// TIA Portal V16 export
// export: Created 2024-05-17T05:47:00.9022411Z, ExportSetting WithDefaults, DisplayName Totally Integrated Automation Portal, DisplayVersion V16, DisplayName TIA Portal Version Control Interface, DisplayVersion V16, DisplayName TIA Portal Openness, DisplayVersion V16, DisplayName STEP 7 Professional, DisplayVersion V16, DisplayName STEP 7 Safety, DisplayVersion V16, DisplayName WinCC Professional, DisplayVersion V16
FUNCTION_BLOCK "K03_状态"   // FB3, LAD
{ S7_Optimized_Access := 'TRUE' }
VERSION : 0.1
// stored: AutoNumber false, IsIECCheckEnabled false, IsRetainMemResEnabled false, MemoryReserve 100, SetENOAutomatically false, UDAEnableTagReadback false
   VAR
      放行延迟 : IEC_TIMER;
   END_VAR
   VAR_TEMP
      M_Pluse : Array[1..20] of Bool;
   END_VAR
   VAR_TEMP   // added for the SCL form of the ladder/FBD networks
      _w1 : Bool;
      _w2 : Bool;
      _w3 : Bool;
      _w4 : Bool;
      _w5 : Bool;
      _w6 : Bool;
      _w7 : Bool;
      _w8 : Bool;
      _w9 : Bool;
      _w10 : Bool;
      _w11 : Bool;
      _w12 : Bool;
      _w13 : Bool;
      _w14 : Bool;
      _w15 : Bool;
   END_VAR
BEGIN

REGION Network 1: 初始2s
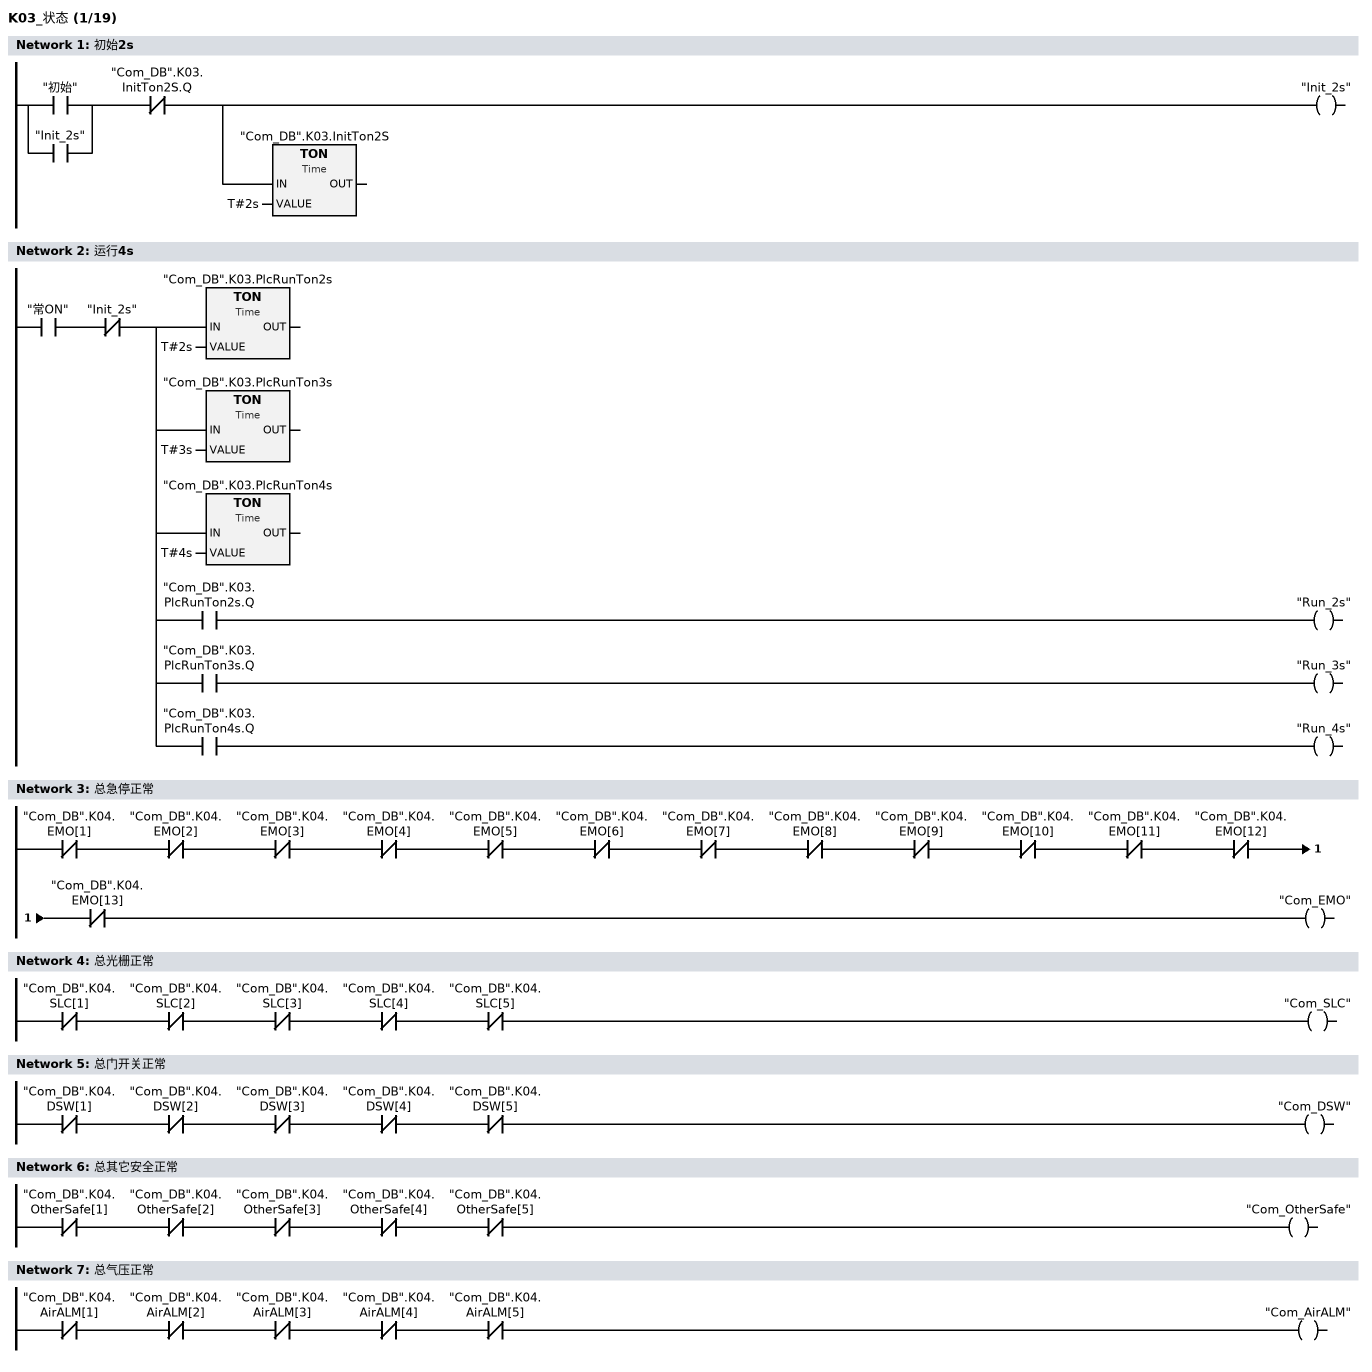
   "Init_2s" := ("初始" OR "Init_2s") AND NOT "Com_DB".K03.InitTon2S.Q;
   "Com_DB".K03.InitTon2S.TON(IN := "Init_2s", PT := T#2s);   // TON coil
END_REGION

REGION Network 2: 运行4s
   #_w1 := "常ON" AND NOT "Init_2s";
   "Com_DB".K03.PlcRunTon2s.TON(IN := #_w1, PT := T#2s);   // TON coil
   "Com_DB".K03.PlcRunTon3s.TON(IN := #_w1, PT := T#3s);   // TON coil
   "Com_DB".K03.PlcRunTon4s.TON(IN := #_w1, PT := T#4s);   // TON coil
   "Run_2s" := #_w1 AND "Com_DB".K03.PlcRunTon2s.Q;
   "Run_3s" := #_w1 AND "Com_DB".K03.PlcRunTon3s.Q;
   "Run_4s" := #_w1 AND "Com_DB".K03.PlcRunTon4s.Q;
END_REGION

REGION Network 3: 总急停正常
   RUNG wire#powerrail
      I_Contact( "Com_DB".K04.EMO[1] )
      I_Contact( "Com_DB".K04.EMO[2] )
      I_Contact( "Com_DB".K04.EMO[3] )
      I_Contact( "Com_DB".K04.EMO[4] )
      I_Contact( "Com_DB".K04.EMO[5] )
      I_Contact( "Com_DB".K04.EMO[6] )
      I_Contact( "Com_DB".K04.EMO[7] )
      I_Contact( "Com_DB".K04.EMO[8] )
      I_Contact( "Com_DB".K04.EMO[9] )
      I_Contact( "Com_DB".K04.EMO[10] )
      I_Contact( "Com_DB".K04.EMO[11] )
      I_Contact( "Com_DB".K04.EMO[12] )
      I_Contact( "Com_DB".K04.EMO[13] )
      Coil( "Com_EMO" )
   END_RUNG
   // the same network as SCL:
   "Com_EMO" := NOT "Com_DB".K04.EMO[1] AND NOT "Com_DB".K04.EMO[2] AND NOT "Com_DB".K04.EMO[3] AND NOT "Com_DB".K04.EMO[4] AND NOT "Com_DB".K04.EMO[5] AND NOT "Com_DB".K04.EMO[6] AND NOT "Com_DB".K04.EMO[7] AND NOT "Com_DB".K04.EMO[8] AND NOT "Com_DB".K04.EMO[9] AND NOT "Com_DB".K04.EMO[10] AND NOT "Com_DB".K04.EMO[11] AND NOT "Com_DB".K04.EMO[12] AND NOT "Com_DB".K04.EMO[13];
END_REGION

REGION Network 4: 总光栅正常
   RUNG wire#powerrail
      I_Contact( "Com_DB".K04.SLC[1] )
      I_Contact( "Com_DB".K04.SLC[2] )
      I_Contact( "Com_DB".K04.SLC[3] )
      I_Contact( "Com_DB".K04.SLC[4] )
      I_Contact( "Com_DB".K04.SLC[5] )
      Coil( "Com_SLC" )
   END_RUNG
   // the same network as SCL:
   "Com_SLC" := NOT "Com_DB".K04.SLC[1] AND NOT "Com_DB".K04.SLC[2] AND NOT "Com_DB".K04.SLC[3] AND NOT "Com_DB".K04.SLC[4] AND NOT "Com_DB".K04.SLC[5];
END_REGION

REGION Network 5: 总门开关正常
   RUNG wire#powerrail
      I_Contact( "Com_DB".K04.DSW[1] )
      I_Contact( "Com_DB".K04.DSW[2] )
      I_Contact( "Com_DB".K04.DSW[3] )
      I_Contact( "Com_DB".K04.DSW[4] )
      I_Contact( "Com_DB".K04.DSW[5] )
      Coil( "Com_DSW" )
   END_RUNG
   // the same network as SCL:
   "Com_DSW" := NOT "Com_DB".K04.DSW[1] AND NOT "Com_DB".K04.DSW[2] AND NOT "Com_DB".K04.DSW[3] AND NOT "Com_DB".K04.DSW[4] AND NOT "Com_DB".K04.DSW[5];
END_REGION

REGION Network 6: 总其它安全正常
   RUNG wire#powerrail
      I_Contact( "Com_DB".K04.OtherSafe[1] )
      I_Contact( "Com_DB".K04.OtherSafe[2] )
      I_Contact( "Com_DB".K04.OtherSafe[3] )
      I_Contact( "Com_DB".K04.OtherSafe[4] )
      I_Contact( "Com_DB".K04.OtherSafe[5] )
      Coil( "Com_OtherSafe" )
   END_RUNG
   // the same network as SCL:
   "Com_OtherSafe" := NOT "Com_DB".K04.OtherSafe[1] AND NOT "Com_DB".K04.OtherSafe[2] AND NOT "Com_DB".K04.OtherSafe[3] AND NOT "Com_DB".K04.OtherSafe[4] AND NOT "Com_DB".K04.OtherSafe[5];
END_REGION

REGION Network 7: 总气压正常
   RUNG wire#powerrail
      I_Contact( "Com_DB".K04.AirALM[1] )
      I_Contact( "Com_DB".K04.AirALM[2] )
      I_Contact( "Com_DB".K04.AirALM[3] )
      I_Contact( "Com_DB".K04.AirALM[4] )
      I_Contact( "Com_DB".K04.AirALM[5] )
      Coil( "Com_AirALM" )
   END_RUNG
   // the same network as SCL:
   "Com_AirALM" := NOT "Com_DB".K04.AirALM[1] AND NOT "Com_DB".K04.AirALM[2] AND NOT "Com_DB".K04.AirALM[3] AND NOT "Com_DB".K04.AirALM[4] AND NOT "Com_DB".K04.AirALM[5];
END_REGION

REGION Network 8: EN传感器滤波
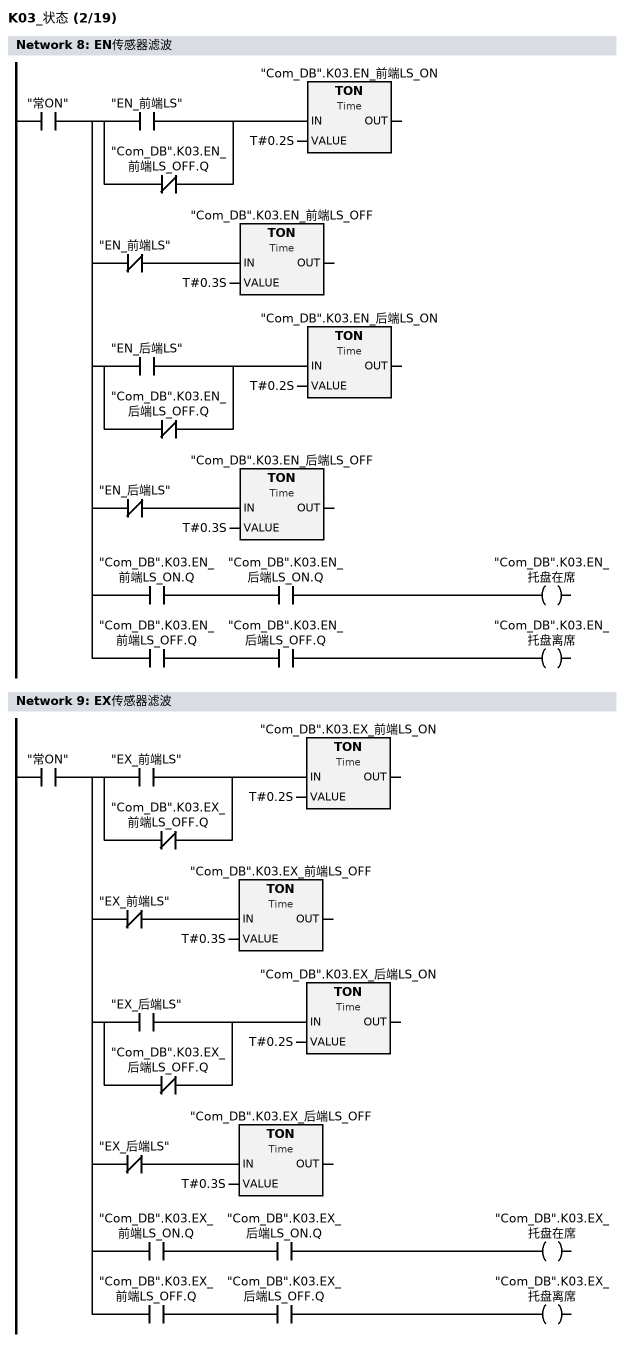
   "Com_DB".K03.EN_前端LS_ON.TON(IN := "常ON" AND ("EN_前端LS" OR NOT "Com_DB".K03.EN_前端LS_OFF.Q), PT := T#0.2S);   // TON coil
   "Com_DB".K03.EN_前端LS_OFF.TON(IN := "常ON" AND NOT "EN_前端LS", PT := T#0.3S);   // TON coil
   "Com_DB".K03.EN_后端LS_ON.TON(IN := "常ON" AND ("EN_后端LS" OR NOT "Com_DB".K03.EN_后端LS_OFF.Q), PT := T#0.2S);   // TON coil
   "Com_DB".K03.EN_后端LS_OFF.TON(IN := "常ON" AND NOT "EN_后端LS", PT := T#0.3S);   // TON coil
   "Com_DB".K03.EN_托盘在席 := "常ON" AND "Com_DB".K03.EN_前端LS_ON.Q AND "Com_DB".K03.EN_后端LS_ON.Q;
   "Com_DB".K03.EN_托盘离席 := "常ON" AND "Com_DB".K03.EN_前端LS_OFF.Q AND "Com_DB".K03.EN_后端LS_OFF.Q;
END_REGION

REGION Network 9: EX传感器滤波
   "Com_DB".K03.EX_前端LS_ON.TON(IN := "常ON" AND ("EX_前端LS" OR NOT "Com_DB".K03.EX_前端LS_OFF.Q), PT := T#0.2S);   // TON coil
   "Com_DB".K03.EX_前端LS_OFF.TON(IN := "常ON" AND NOT "EX_前端LS", PT := T#0.3S);   // TON coil
   "Com_DB".K03.EX_后端LS_ON.TON(IN := "常ON" AND ("EX_后端LS" OR NOT "Com_DB".K03.EX_后端LS_OFF.Q), PT := T#0.2S);   // TON coil
   "Com_DB".K03.EX_后端LS_OFF.TON(IN := "常ON" AND NOT "EX_后端LS", PT := T#0.3S);   // TON coil
   "Com_DB".K03.EX_托盘在席 := "常ON" AND "Com_DB".K03.EX_前端LS_ON.Q AND "Com_DB".K03.EX_后端LS_ON.Q;
   "Com_DB".K03.EX_托盘离席 := "常ON" AND "Com_DB".K03.EX_前端LS_OFF.Q AND "Com_DB".K03.EX_后端LS_OFF.Q;
END_REGION

REGION Network 10: ST01上层传感器滤波
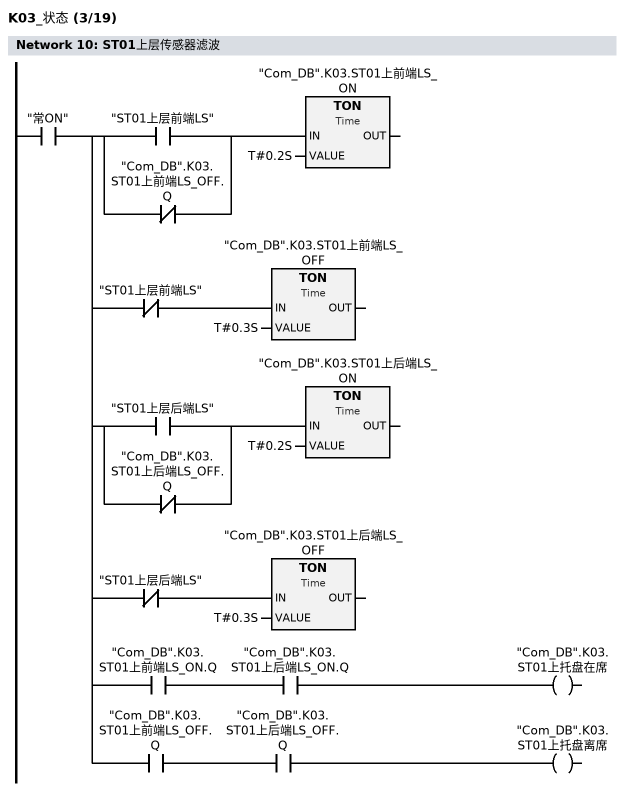
   "Com_DB".K03.ST01上前端LS_ON.TON(IN := "常ON" AND ("ST01上层前端LS" OR NOT "Com_DB".K03.ST01上前端LS_OFF.Q), PT := T#0.2S);   // TON coil
   "Com_DB".K03.ST01上前端LS_OFF.TON(IN := "常ON" AND NOT "ST01上层前端LS", PT := T#0.3S);   // TON coil
   "Com_DB".K03.ST01上后端LS_ON.TON(IN := "常ON" AND ("ST01上层后端LS" OR NOT "Com_DB".K03.ST01上后端LS_OFF.Q), PT := T#0.2S);   // TON coil
   "Com_DB".K03.ST01上后端LS_OFF.TON(IN := "常ON" AND NOT "ST01上层后端LS", PT := T#0.3S);   // TON coil
   "Com_DB".K03.ST01上托盘在席 := "常ON" AND "Com_DB".K03.ST01上前端LS_ON.Q AND "Com_DB".K03.ST01上后端LS_ON.Q;
   "Com_DB".K03.ST01上托盘离席 := "常ON" AND "Com_DB".K03.ST01上前端LS_OFF.Q AND "Com_DB".K03.ST01上后端LS_OFF.Q;
END_REGION

REGION Network 11: ST01下层传感器滤波
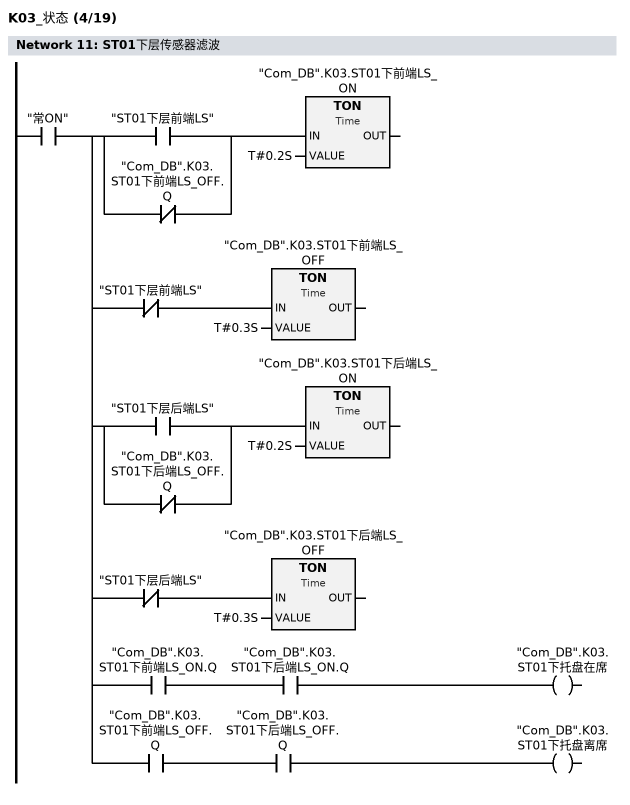
   "Com_DB".K03.ST01下前端LS_ON.TON(IN := "常ON" AND ("ST01下层前端LS" OR NOT "Com_DB".K03.ST01下前端LS_OFF.Q), PT := T#0.2S);   // TON coil
   "Com_DB".K03.ST01下前端LS_OFF.TON(IN := "常ON" AND NOT "ST01下层前端LS", PT := T#0.3S);   // TON coil
   "Com_DB".K03.ST01下后端LS_ON.TON(IN := "常ON" AND ("ST01下层后端LS" OR NOT "Com_DB".K03.ST01下后端LS_OFF.Q), PT := T#0.2S);   // TON coil
   "Com_DB".K03.ST01下后端LS_OFF.TON(IN := "常ON" AND NOT "ST01下层后端LS", PT := T#0.3S);   // TON coil
   "Com_DB".K03.ST01下托盘在席 := "常ON" AND "Com_DB".K03.ST01下前端LS_ON.Q AND "Com_DB".K03.ST01下后端LS_ON.Q;
   "Com_DB".K03.ST01下托盘离席 := "常ON" AND "Com_DB".K03.ST01下前端LS_OFF.Q AND "Com_DB".K03.ST01下后端LS_OFF.Q;
END_REGION

REGION Network 12: ST02上层传感器滤波
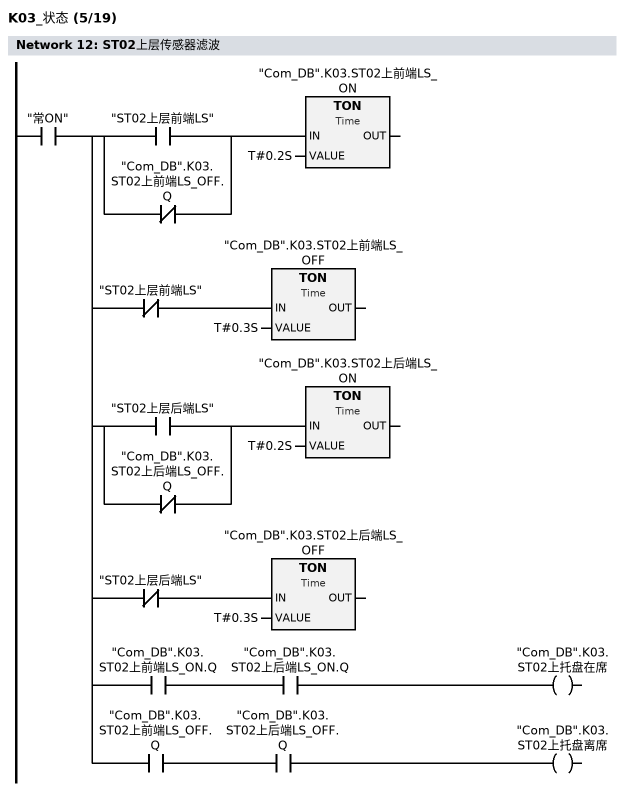
   "Com_DB".K03.ST02上前端LS_ON.TON(IN := "常ON" AND ("ST02上层前端LS" OR NOT "Com_DB".K03.ST02上前端LS_OFF.Q), PT := T#0.2S);   // TON coil
   "Com_DB".K03.ST02上前端LS_OFF.TON(IN := "常ON" AND NOT "ST02上层前端LS", PT := T#0.3S);   // TON coil
   "Com_DB".K03.ST02上后端LS_ON.TON(IN := "常ON" AND ("ST02上层后端LS" OR NOT "Com_DB".K03.ST02上后端LS_OFF.Q), PT := T#0.2S);   // TON coil
   "Com_DB".K03.ST02上后端LS_OFF.TON(IN := "常ON" AND NOT "ST02上层后端LS", PT := T#0.3S);   // TON coil
   "Com_DB".K03.ST02上托盘在席 := "常ON" AND "Com_DB".K03.ST02上前端LS_ON.Q AND "Com_DB".K03.ST02上后端LS_ON.Q;
   "Com_DB".K03.ST02上托盘离席 := "常ON" AND "Com_DB".K03.ST02上前端LS_OFF.Q AND "Com_DB".K03.ST02上后端LS_OFF.Q;
END_REGION

REGION Network 13: ST02下层传感器滤波
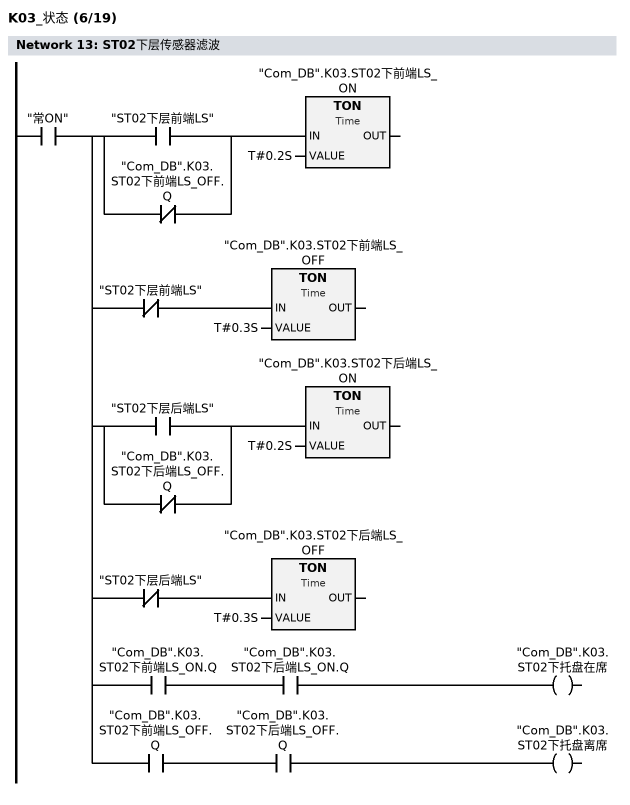
   "Com_DB".K03.ST02下前端LS_ON.TON(IN := "常ON" AND ("ST02下层前端LS" OR NOT "Com_DB".K03.ST02下前端LS_OFF.Q), PT := T#0.2S);   // TON coil
   "Com_DB".K03.ST02下前端LS_OFF.TON(IN := "常ON" AND NOT "ST02下层前端LS", PT := T#0.3S);   // TON coil
   "Com_DB".K03.ST02下后端LS_ON.TON(IN := "常ON" AND ("ST02下层后端LS" OR NOT "Com_DB".K03.ST02下后端LS_OFF.Q), PT := T#0.2S);   // TON coil
   "Com_DB".K03.ST02下后端LS_OFF.TON(IN := "常ON" AND NOT "ST02下层后端LS", PT := T#0.3S);   // TON coil
   "Com_DB".K03.ST02下托盘在席 := "常ON" AND "Com_DB".K03.ST02下前端LS_ON.Q AND "Com_DB".K03.ST02下后端LS_ON.Q;
   "Com_DB".K03.ST02下托盘离席 := "常ON" AND "Com_DB".K03.ST02下前端LS_OFF.Q AND "Com_DB".K03.ST02下后端LS_OFF.Q;
END_REGION

REGION Network 14: ST03上层传感器滤波
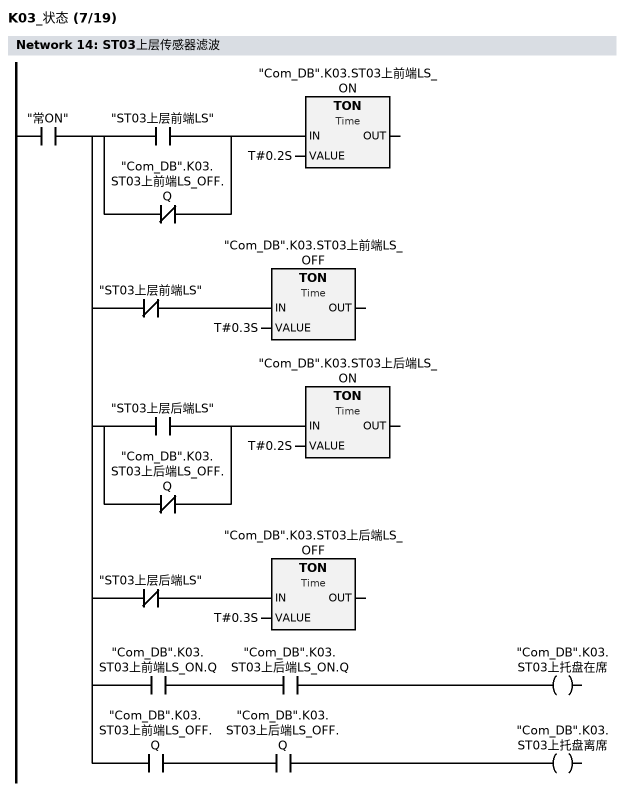
   "Com_DB".K03.ST03上前端LS_ON.TON(IN := "常ON" AND ("ST03上层前端LS" OR NOT "Com_DB".K03.ST03上前端LS_OFF.Q), PT := T#0.2S);   // TON coil
   "Com_DB".K03.ST03上前端LS_OFF.TON(IN := "常ON" AND NOT "ST03上层前端LS", PT := T#0.3S);   // TON coil
   "Com_DB".K03.ST03上后端LS_ON.TON(IN := "常ON" AND ("ST03上层后端LS" OR NOT "Com_DB".K03.ST03上后端LS_OFF.Q), PT := T#0.2S);   // TON coil
   "Com_DB".K03.ST03上后端LS_OFF.TON(IN := "常ON" AND NOT "ST03上层后端LS", PT := T#0.3S);   // TON coil
   "Com_DB".K03.ST03上托盘在席 := "常ON" AND "Com_DB".K03.ST03上前端LS_ON.Q AND "Com_DB".K03.ST03上后端LS_ON.Q;
   "Com_DB".K03.ST03上托盘离席 := "常ON" AND "Com_DB".K03.ST03上前端LS_OFF.Q AND "Com_DB".K03.ST03上后端LS_OFF.Q;
END_REGION

REGION Network 15: ST03下层传感器滤波
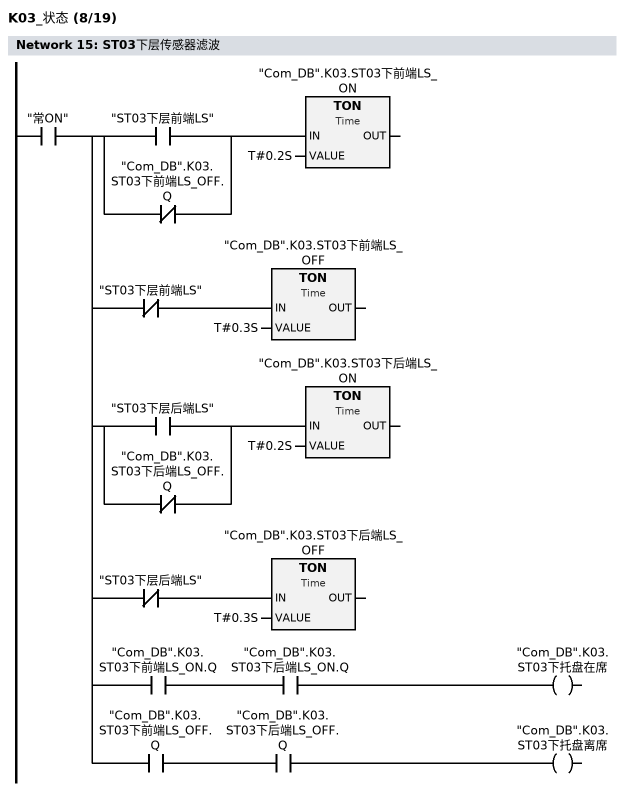
   "Com_DB".K03.ST03下前端LS_ON.TON(IN := "常ON" AND ("ST03下层前端LS" OR NOT "Com_DB".K03.ST03下前端LS_OFF.Q), PT := T#0.2S);   // TON coil
   "Com_DB".K03.ST03下前端LS_OFF.TON(IN := "常ON" AND NOT "ST03下层前端LS", PT := T#0.3S);   // TON coil
   "Com_DB".K03.ST03下后端LS_ON.TON(IN := "常ON" AND ("ST03下层后端LS" OR NOT "Com_DB".K03.ST03下后端LS_OFF.Q), PT := T#0.2S);   // TON coil
   "Com_DB".K03.ST03下后端LS_OFF.TON(IN := "常ON" AND NOT "ST03下层后端LS", PT := T#0.3S);   // TON coil
   "Com_DB".K03.ST03下托盘在席 := "常ON" AND "Com_DB".K03.ST03下前端LS_ON.Q AND "Com_DB".K03.ST03下后端LS_ON.Q;
   "Com_DB".K03.ST03下托盘离席 := "常ON" AND "Com_DB".K03.ST03下前端LS_OFF.Q AND "Com_DB".K03.ST03下后端LS_OFF.Q;
END_REGION

REGION Network 16: ST04上层传感器滤波
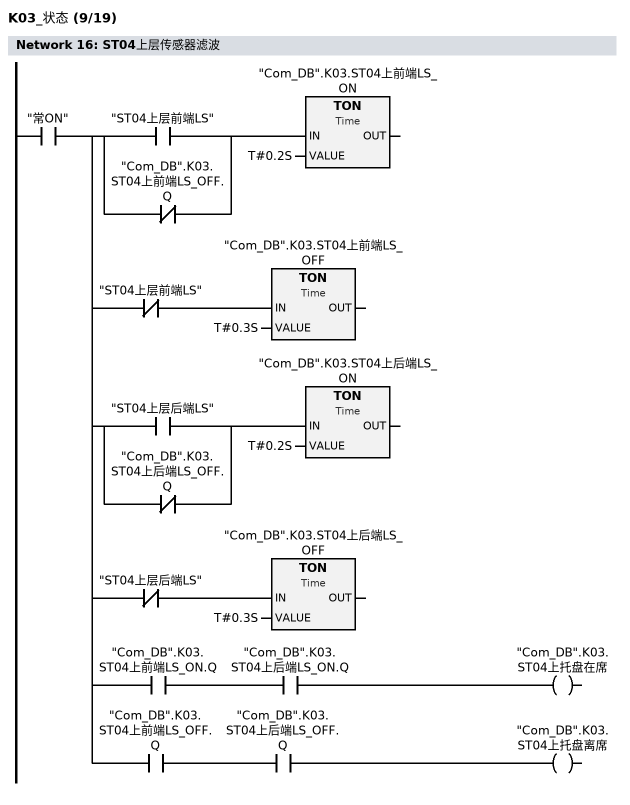
   "Com_DB".K03.ST04上前端LS_ON.TON(IN := "常ON" AND ("ST04上层前端LS" OR NOT "Com_DB".K03.ST04上前端LS_OFF.Q), PT := T#0.2S);   // TON coil
   "Com_DB".K03.ST04上前端LS_OFF.TON(IN := "常ON" AND NOT "ST04上层前端LS", PT := T#0.3S);   // TON coil
   "Com_DB".K03.ST04上后端LS_ON.TON(IN := "常ON" AND ("ST04上层后端LS" OR NOT "Com_DB".K03.ST04上后端LS_OFF.Q), PT := T#0.2S);   // TON coil
   "Com_DB".K03.ST04上后端LS_OFF.TON(IN := "常ON" AND NOT "ST04上层后端LS", PT := T#0.3S);   // TON coil
   "Com_DB".K03.ST04上托盘在席 := "常ON" AND "Com_DB".K03.ST04上前端LS_ON.Q AND "Com_DB".K03.ST04上后端LS_ON.Q;
   "Com_DB".K03.ST04上托盘离席 := "常ON" AND "Com_DB".K03.ST04上前端LS_OFF.Q AND "Com_DB".K03.ST04上后端LS_OFF.Q;
END_REGION

REGION Network 17: ST05上层传感器滤波
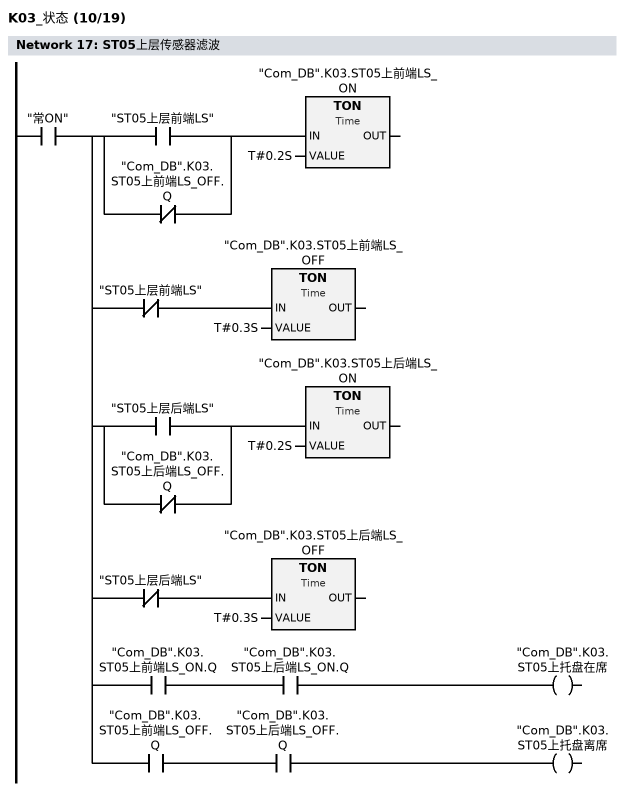
   "Com_DB".K03.ST05上前端LS_ON.TON(IN := "常ON" AND ("ST05上层前端LS" OR NOT "Com_DB".K03.ST05上前端LS_OFF.Q), PT := T#0.2S);   // TON coil
   "Com_DB".K03.ST05上前端LS_OFF.TON(IN := "常ON" AND NOT "ST05上层前端LS", PT := T#0.3S);   // TON coil
   "Com_DB".K03.ST05上后端LS_ON.TON(IN := "常ON" AND ("ST05上层后端LS" OR NOT "Com_DB".K03.ST05上后端LS_OFF.Q), PT := T#0.2S);   // TON coil
   "Com_DB".K03.ST05上后端LS_OFF.TON(IN := "常ON" AND NOT "ST05上层后端LS", PT := T#0.3S);   // TON coil
   "Com_DB".K03.ST05上托盘在席 := "常ON" AND "Com_DB".K03.ST05上前端LS_ON.Q AND "Com_DB".K03.ST05上后端LS_ON.Q;
   "Com_DB".K03.ST05上托盘离席 := "常ON" AND "Com_DB".K03.ST05上前端LS_OFF.Q AND "Com_DB".K03.ST05上后端LS_OFF.Q;
END_REGION

REGION Network 18: ST06上层传感器滤波
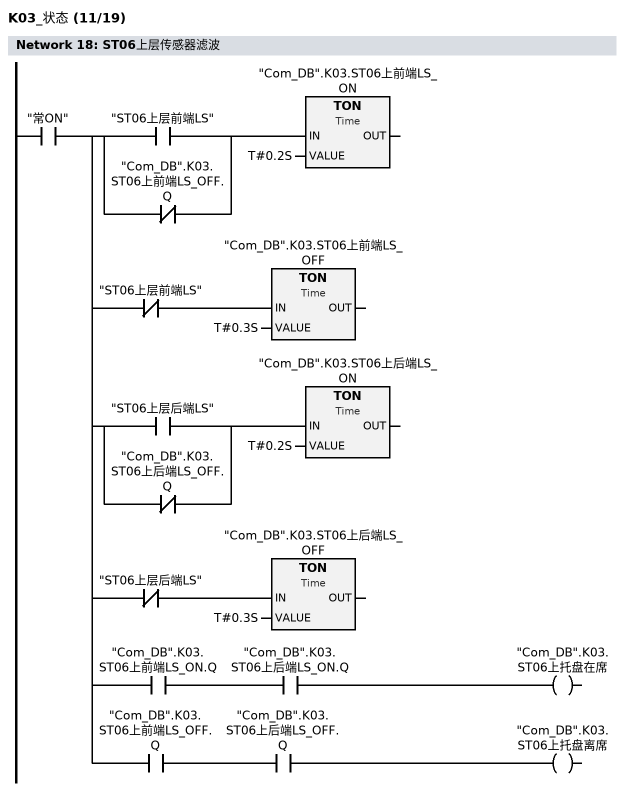
   "Com_DB".K03.ST06上前端LS_ON.TON(IN := "常ON" AND ("ST06上层前端LS" OR NOT "Com_DB".K03.ST06上前端LS_OFF.Q), PT := T#0.2S);   // TON coil
   "Com_DB".K03.ST06上前端LS_OFF.TON(IN := "常ON" AND NOT "ST06上层前端LS", PT := T#0.3S);   // TON coil
   "Com_DB".K03.ST06上后端LS_ON.TON(IN := "常ON" AND ("ST06上层后端LS" OR NOT "Com_DB".K03.ST06上后端LS_OFF.Q), PT := T#0.2S);   // TON coil
   "Com_DB".K03.ST06上后端LS_OFF.TON(IN := "常ON" AND NOT "ST06上层后端LS", PT := T#0.3S);   // TON coil
   "Com_DB".K03.ST06上托盘在席 := "常ON" AND "Com_DB".K03.ST06上前端LS_ON.Q AND "Com_DB".K03.ST06上后端LS_ON.Q;
   "Com_DB".K03.ST06上托盘离席 := "常ON" AND "Com_DB".K03.ST06上前端LS_OFF.Q AND "Com_DB".K03.ST06上后端LS_OFF.Q;
END_REGION

REGION Network 19: ST07上层传感器滤波
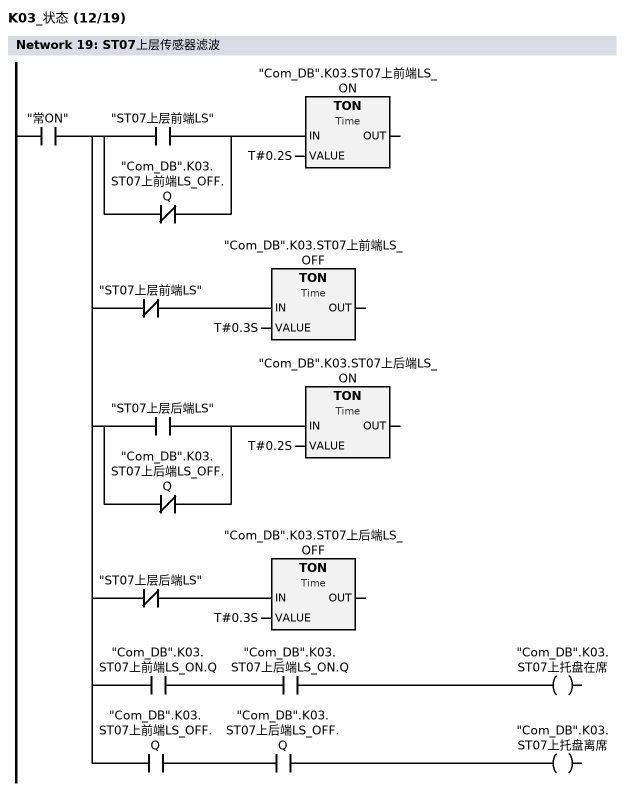
   "Com_DB".K03.ST07上前端LS_ON.TON(IN := "常ON" AND ("ST07上层前端LS" OR NOT "Com_DB".K03.ST07上前端LS_OFF.Q), PT := T#0.2S);   // TON coil
   "Com_DB".K03.ST07上前端LS_OFF.TON(IN := "常ON" AND NOT "ST07上层前端LS", PT := T#0.3S);   // TON coil
   "Com_DB".K03.ST07上后端LS_ON.TON(IN := "常ON" AND ("ST07上层后端LS" OR NOT "Com_DB".K03.ST07上后端LS_OFF.Q), PT := T#0.2S);   // TON coil
   "Com_DB".K03.ST07上后端LS_OFF.TON(IN := "常ON" AND NOT "ST07上层后端LS", PT := T#0.3S);   // TON coil
   "Com_DB".K03.ST07上托盘在席 := "常ON" AND "Com_DB".K03.ST07上前端LS_ON.Q AND "Com_DB".K03.ST07上后端LS_ON.Q;
   "Com_DB".K03.ST07上托盘离席 := "常ON" AND "Com_DB".K03.ST07上前端LS_OFF.Q AND "Com_DB".K03.ST07上后端LS_OFF.Q;
END_REGION

REGION Network 20: ST08上层传感器滤波
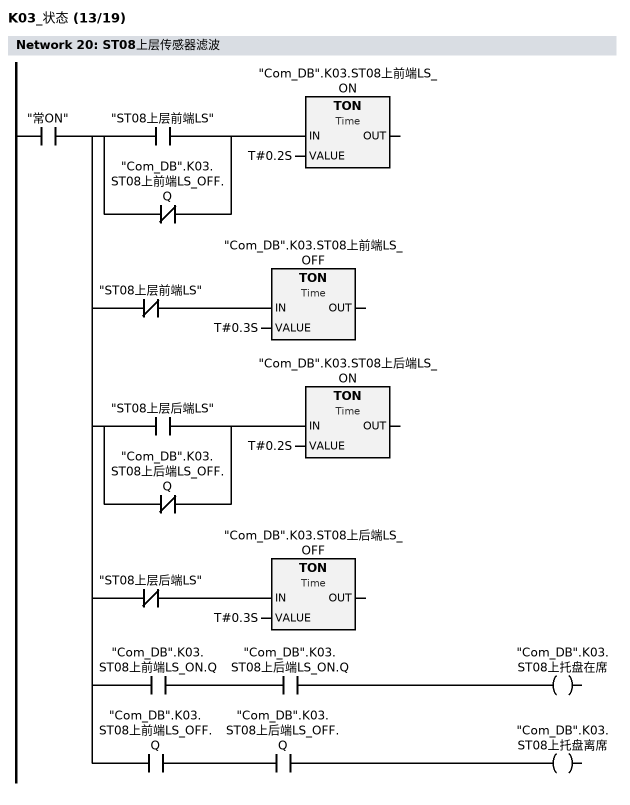
   "Com_DB".K03.ST08上前端LS_ON.TON(IN := "常ON" AND ("ST08上层前端LS" OR NOT "Com_DB".K03.ST08上前端LS_OFF.Q), PT := T#0.2S);   // TON coil
   "Com_DB".K03.ST08上前端LS_OFF.TON(IN := "常ON" AND NOT "ST08上层前端LS", PT := T#0.3S);   // TON coil
   "Com_DB".K03.ST08上后端LS_ON.TON(IN := "常ON" AND ("ST08上层后端LS" OR NOT "Com_DB".K03.ST08上后端LS_OFF.Q), PT := T#0.2S);   // TON coil
   "Com_DB".K03.ST08上后端LS_OFF.TON(IN := "常ON" AND NOT "ST08上层后端LS", PT := T#0.3S);   // TON coil
   "Com_DB".K03.ST08上托盘在席 := "常ON" AND "Com_DB".K03.ST08上前端LS_ON.Q AND "Com_DB".K03.ST08上后端LS_ON.Q;
   "Com_DB".K03.ST08上托盘离席 := "常ON" AND "Com_DB".K03.ST08上前端LS_OFF.Q AND "Com_DB".K03.ST08上后端LS_OFF.Q;
END_REGION

REGION Network 21: ST09上层传感器滤波
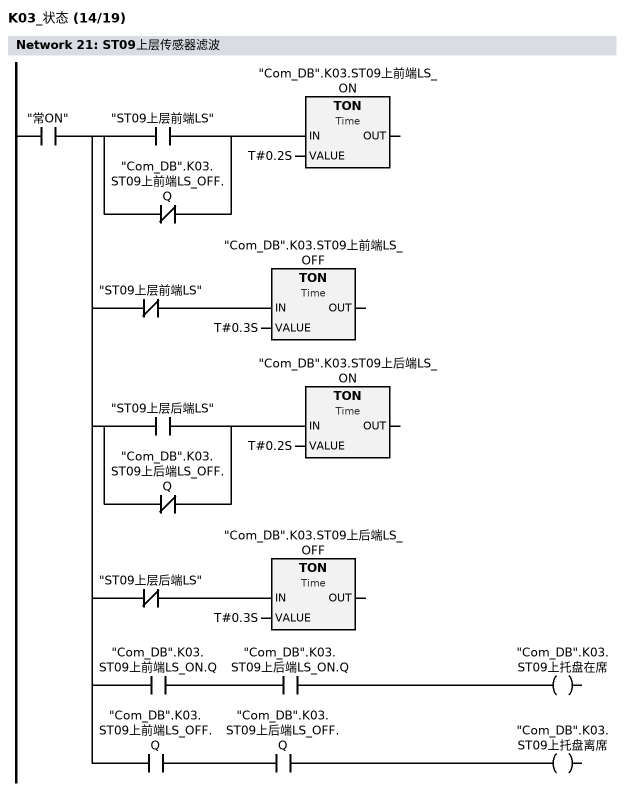
   "Com_DB".K03.ST09上前端LS_ON.TON(IN := "常ON" AND ("ST09上层前端LS" OR NOT "Com_DB".K03.ST09上前端LS_OFF.Q), PT := T#0.2S);   // TON coil
   "Com_DB".K03.ST09上前端LS_OFF.TON(IN := "常ON" AND NOT "ST09上层前端LS", PT := T#0.3S);   // TON coil
   "Com_DB".K03.ST09上后端LS_ON.TON(IN := "常ON" AND ("ST09上层后端LS" OR NOT "Com_DB".K03.ST09上后端LS_OFF.Q), PT := T#0.2S);   // TON coil
   "Com_DB".K03.ST09上后端LS_OFF.TON(IN := "常ON" AND NOT "ST09上层后端LS", PT := T#0.3S);   // TON coil
   "Com_DB".K03.ST09上托盘在席 := "常ON" AND "Com_DB".K03.ST09上前端LS_ON.Q AND "Com_DB".K03.ST09上后端LS_ON.Q;
   "Com_DB".K03.ST09上托盘离席 := "常ON" AND "Com_DB".K03.ST09上前端LS_OFF.Q AND "Com_DB".K03.ST09上后端LS_OFF.Q;
END_REGION

REGION Network 22: ST10上层传感器滤波
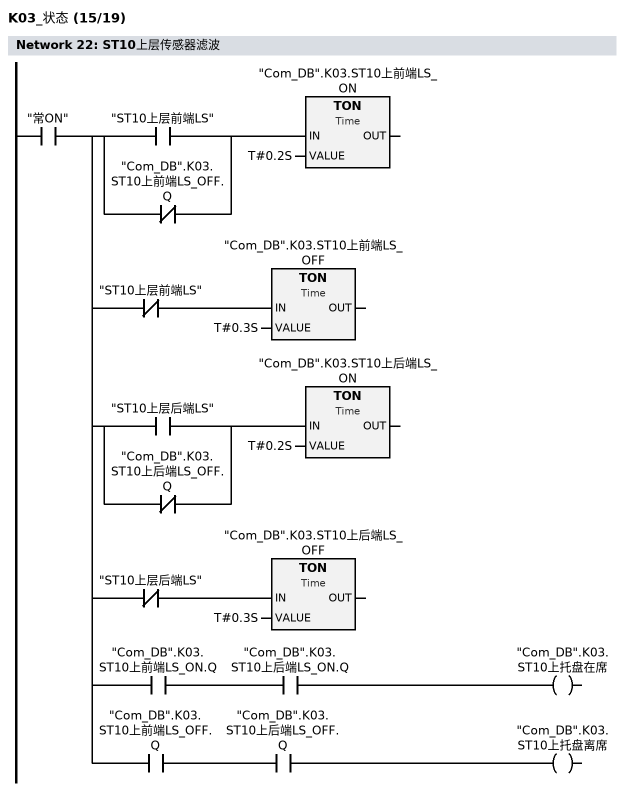
   "Com_DB".K03.ST10上前端LS_ON.TON(IN := "常ON" AND ("ST10上层前端LS" OR NOT "Com_DB".K03.ST10上前端LS_OFF.Q), PT := T#0.2S);   // TON coil
   "Com_DB".K03.ST10上前端LS_OFF.TON(IN := "常ON" AND NOT "ST10上层前端LS", PT := T#0.3S);   // TON coil
   "Com_DB".K03.ST10上后端LS_ON.TON(IN := "常ON" AND ("ST10上层后端LS" OR NOT "Com_DB".K03.ST10上后端LS_OFF.Q), PT := T#0.2S);   // TON coil
   "Com_DB".K03.ST10上后端LS_OFF.TON(IN := "常ON" AND NOT "ST10上层后端LS", PT := T#0.3S);   // TON coil
   "Com_DB".K03.ST10上托盘在席 := "常ON" AND "Com_DB".K03.ST10上前端LS_ON.Q AND "Com_DB".K03.ST10上后端LS_ON.Q;
   "Com_DB".K03.ST10上托盘离席 := "常ON" AND "Com_DB".K03.ST10上前端LS_OFF.Q AND "Com_DB".K03.ST10上后端LS_OFF.Q;
END_REGION

REGION Network 23: ST11上层传感器滤波
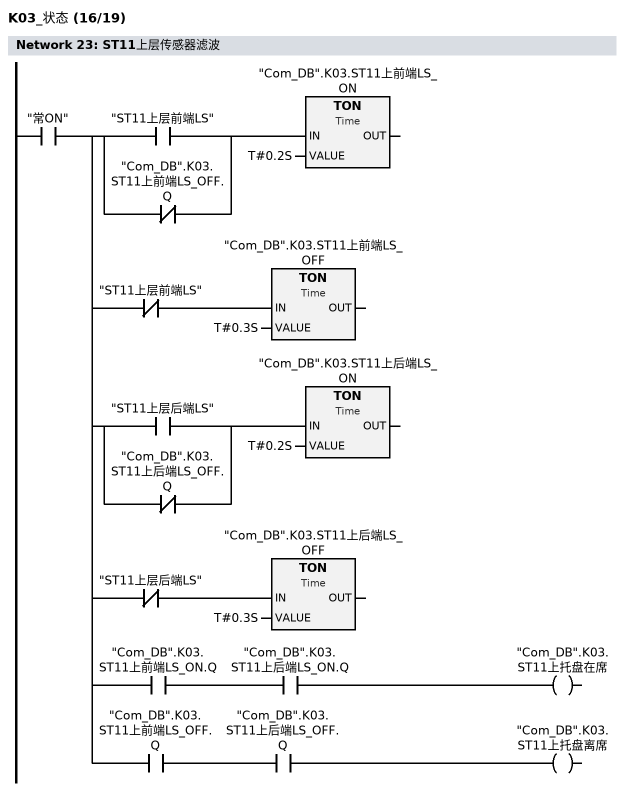
   "Com_DB".K03.ST11上前端LS_ON.TON(IN := "常ON" AND ("ST11上层前端LS" OR NOT "Com_DB".K03.ST11上前端LS_OFF.Q), PT := T#0.2S);   // TON coil
   "Com_DB".K03.ST11上前端LS_OFF.TON(IN := "常ON" AND NOT "ST11上层前端LS", PT := T#0.3S);   // TON coil
   "Com_DB".K03.ST11上后端LS_ON.TON(IN := "常ON" AND ("ST11上层后端LS" OR NOT "Com_DB".K03.ST11上后端LS_OFF.Q), PT := T#0.2S);   // TON coil
   "Com_DB".K03.ST11上后端LS_OFF.TON(IN := "常ON" AND NOT "ST11上层后端LS", PT := T#0.3S);   // TON coil
   "Com_DB".K03.ST11上托盘在席 := "常ON" AND "Com_DB".K03.ST11上前端LS_ON.Q AND "Com_DB".K03.ST11上后端LS_ON.Q;
   "Com_DB".K03.ST11上托盘离席 := "常ON" AND "Com_DB".K03.ST11上前端LS_OFF.Q AND "Com_DB".K03.ST11上后端LS_OFF.Q;
END_REGION

REGION Network 24: ST12上层传感器滤波
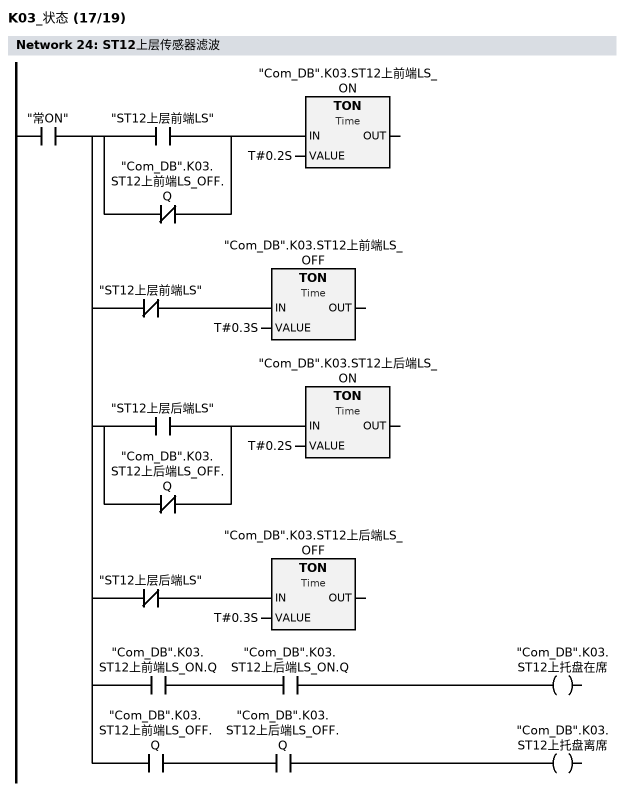
   "Com_DB".K03.ST12上前端LS_ON.TON(IN := "常ON" AND ("ST12上层前端LS" OR NOT "Com_DB".K03.ST12上前端LS_OFF.Q), PT := T#0.2S);   // TON coil
   "Com_DB".K03.ST12上前端LS_OFF.TON(IN := "常ON" AND NOT "ST12上层前端LS", PT := T#0.3S);   // TON coil
   "Com_DB".K03.ST12上后端LS_ON.TON(IN := "常ON" AND ("ST12上层后端LS" OR NOT "Com_DB".K03.ST12上后端LS_OFF.Q), PT := T#0.2S);   // TON coil
   "Com_DB".K03.ST12上后端LS_OFF.TON(IN := "常ON" AND NOT "ST12上层后端LS", PT := T#0.3S);   // TON coil
   "Com_DB".K03.ST12上托盘在席 := "常ON" AND "Com_DB".K03.ST12上前端LS_ON.Q AND "Com_DB".K03.ST12上后端LS_ON.Q;
   "Com_DB".K03.ST12上托盘离席 := "常ON" AND "Com_DB".K03.ST12上前端LS_OFF.Q AND "Com_DB".K03.ST12上后端LS_OFF.Q;
END_REGION

REGION Network 25: ST01-ST12记忆标志
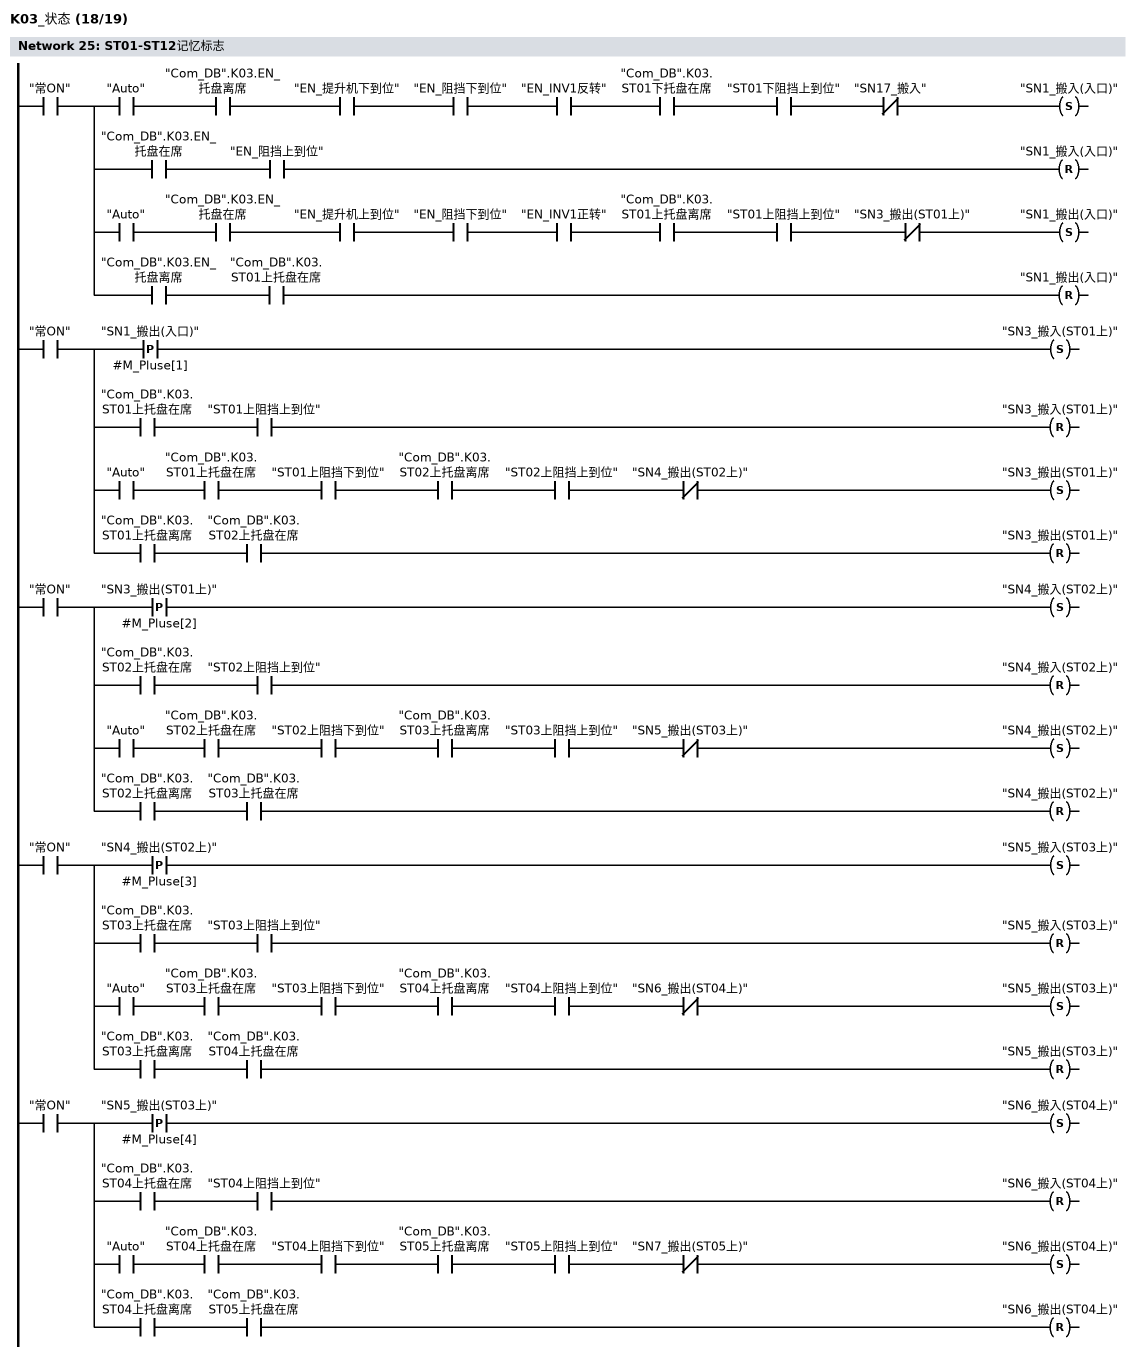
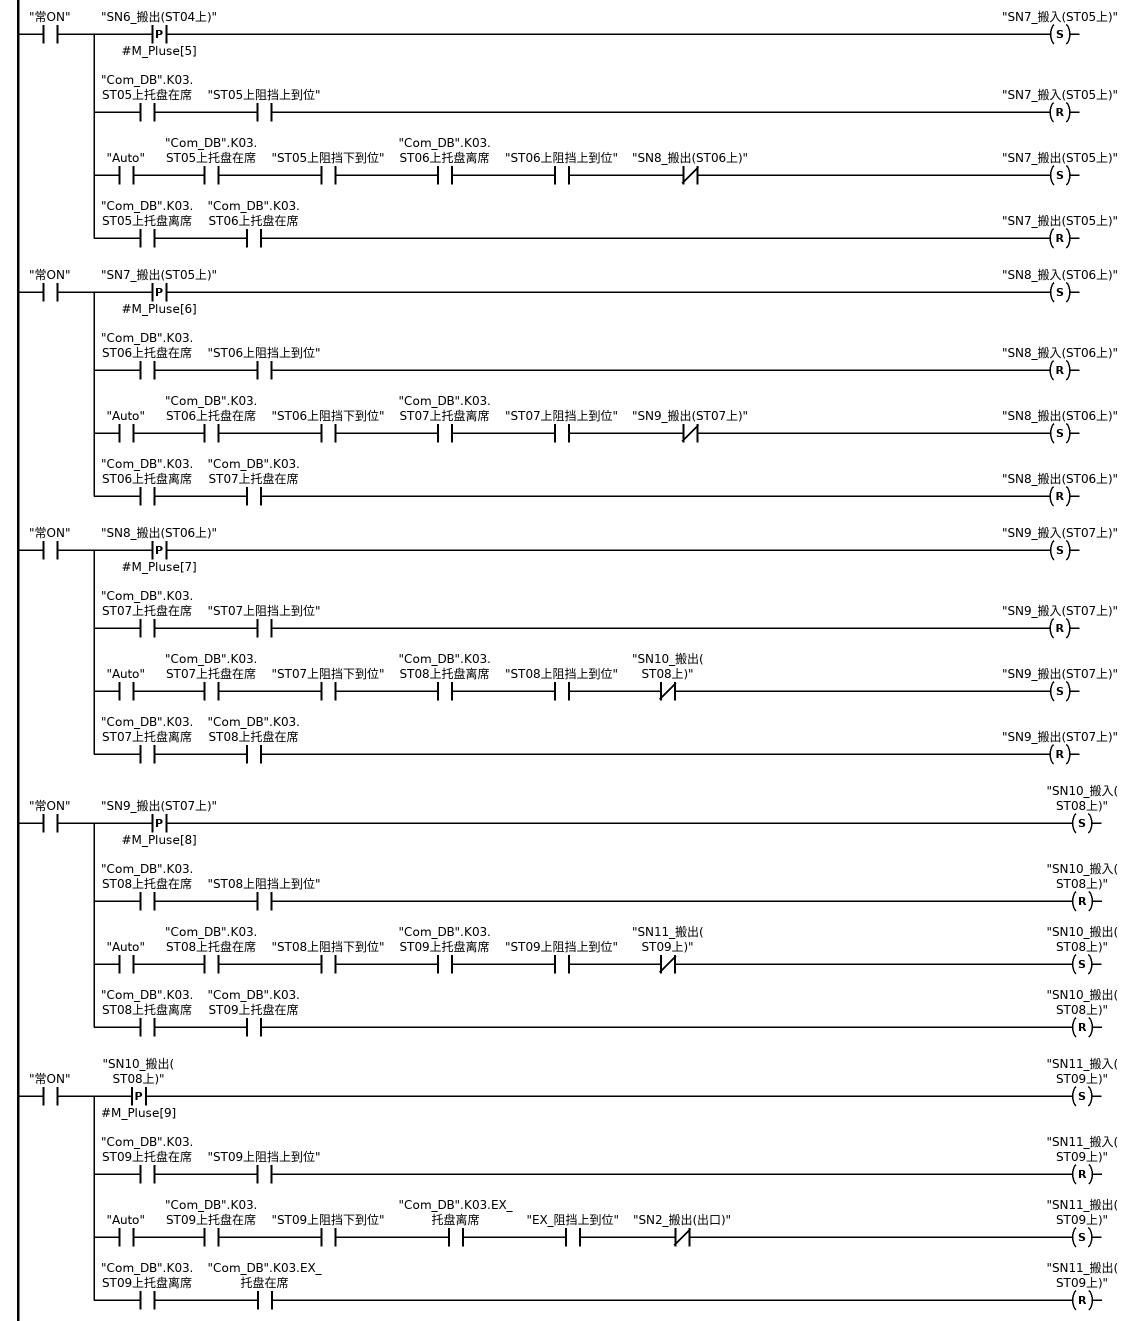
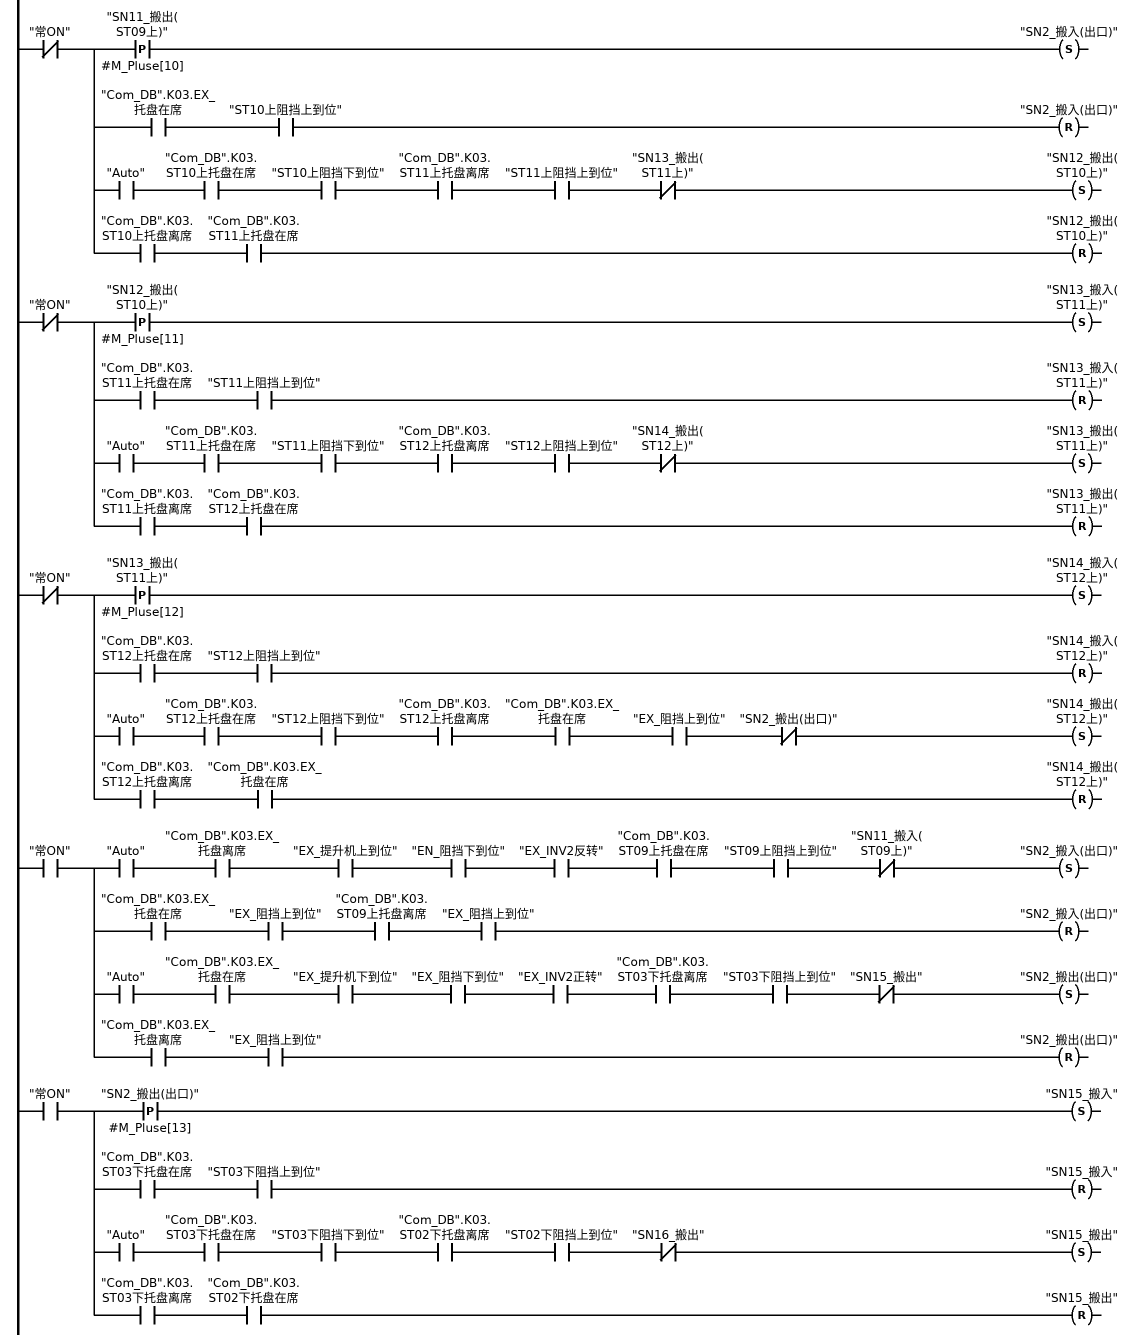
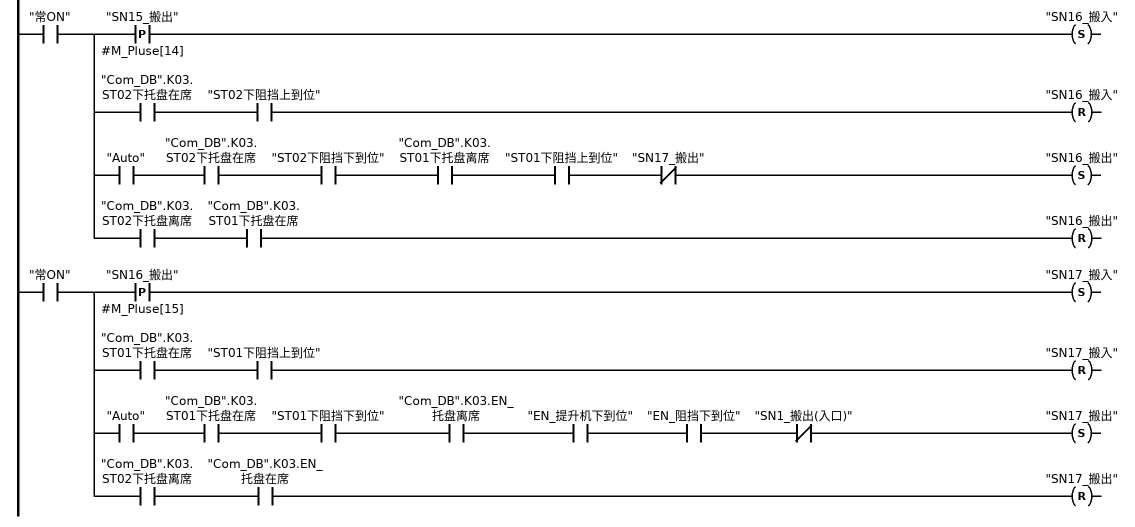
   RUNG wire#powerrail
      Contact( "常ON" )
      wire#w1
      Contact( "Auto" )
      Contact( "Com_DB".K03.EN_托盘离席 )
      Contact( "EN_提升机下到位" )
      Contact( "EN_阻挡下到位" )
      Contact( "EN_INV1反转" )
      Contact( "Com_DB".K03.ST01下托盘在席 )
      Contact( "ST01下阻挡上到位" )
      I_Contact( "SN17_搬入" )
      S_Coil( "SN1_搬入(入口)" )
   END_RUNG
   RUNG wire#w1
      Contact( "Com_DB".K03.EN_托盘在席 )
      Contact( "EN_阻挡上到位" )
      R_Coil( "SN1_搬入(入口)" )
   END_RUNG
   RUNG wire#w1
      Contact( "Auto" )
      Contact( "Com_DB".K03.EN_托盘在席 )
      Contact( "EN_提升机上到位" )
      Contact( "EN_阻挡下到位" )
      Contact( "EN_INV1正转" )
      Contact( "Com_DB".K03.ST01上托盘离席 )
      Contact( "ST01上阻挡上到位" )
      I_Contact( "SN3_搬出(ST01上)" )
      S_Coil( "SN1_搬出(入口)" )
   END_RUNG
   RUNG wire#w1
      Contact( "Com_DB".K03.EN_托盘离席 )
      Contact( "Com_DB".K03.ST01上托盘在席 )
      R_Coil( "SN1_搬出(入口)" )
   END_RUNG
   RUNG wire#powerrail
      Contact( "常ON" )
      wire#w2
      P_Contact(operand := "SN1_搬出(入口)", bit := #M_Pluse[1])
      S_Coil( "SN3_搬入(ST01上)" )
   END_RUNG
   RUNG wire#w2
      Contact( "Com_DB".K03.ST01上托盘在席 )
      Contact( "ST01上阻挡上到位" )
      R_Coil( "SN3_搬入(ST01上)" )
   END_RUNG
   RUNG wire#w2
      Contact( "Auto" )
      Contact( "Com_DB".K03.ST01上托盘在席 )
      Contact( "ST01上阻挡下到位" )
      Contact( "Com_DB".K03.ST02上托盘离席 )
      Contact( "ST02上阻挡上到位" )
      I_Contact( "SN4_搬出(ST02上)" )
      S_Coil( "SN3_搬出(ST01上)" )
   END_RUNG
   RUNG wire#w2
      Contact( "Com_DB".K03.ST01上托盘离席 )
      Contact( "Com_DB".K03.ST02上托盘在席 )
      R_Coil( "SN3_搬出(ST01上)" )
   END_RUNG
   RUNG wire#powerrail
      Contact( "常ON" )
      wire#w3
      P_Contact(operand := "SN3_搬出(ST01上)", bit := #M_Pluse[2])
      S_Coil( "SN4_搬入(ST02上)" )
   END_RUNG
   RUNG wire#w3
      Contact( "Com_DB".K03.ST02上托盘在席 )
      Contact( "ST02上阻挡上到位" )
      R_Coil( "SN4_搬入(ST02上)" )
   END_RUNG
   RUNG wire#w3
      Contact( "Auto" )
      Contact( "Com_DB".K03.ST02上托盘在席 )
      Contact( "ST02上阻挡下到位" )
      Contact( "Com_DB".K03.ST03上托盘离席 )
      Contact( "ST03上阻挡上到位" )
      I_Contact( "SN5_搬出(ST03上)" )
      S_Coil( "SN4_搬出(ST02上)" )
   END_RUNG
   RUNG wire#w3
      Contact( "Com_DB".K03.ST02上托盘离席 )
      Contact( "Com_DB".K03.ST03上托盘在席 )
      R_Coil( "SN4_搬出(ST02上)" )
   END_RUNG
   RUNG wire#powerrail
      Contact( "常ON" )
      wire#w4
      P_Contact(operand := "SN4_搬出(ST02上)", bit := #M_Pluse[3])
      S_Coil( "SN5_搬入(ST03上)" )
   END_RUNG
   RUNG wire#w4
      Contact( "Com_DB".K03.ST03上托盘在席 )
      Contact( "ST03上阻挡上到位" )
      R_Coil( "SN5_搬入(ST03上)" )
   END_RUNG
   RUNG wire#w4
      Contact( "Auto" )
      Contact( "Com_DB".K03.ST03上托盘在席 )
      Contact( "ST03上阻挡下到位" )
      Contact( "Com_DB".K03.ST04上托盘离席 )
      Contact( "ST04上阻挡上到位" )
      I_Contact( "SN6_搬出(ST04上)" )
      S_Coil( "SN5_搬出(ST03上)" )
   END_RUNG
   RUNG wire#w4
      Contact( "Com_DB".K03.ST03上托盘离席 )
      Contact( "Com_DB".K03.ST04上托盘在席 )
      R_Coil( "SN5_搬出(ST03上)" )
   END_RUNG
   RUNG wire#powerrail
      Contact( "常ON" )
      wire#w5
      P_Contact(operand := "SN5_搬出(ST03上)", bit := #M_Pluse[4])
      S_Coil( "SN6_搬入(ST04上)" )
   END_RUNG
   RUNG wire#w5
      Contact( "Com_DB".K03.ST04上托盘在席 )
      Contact( "ST04上阻挡上到位" )
      R_Coil( "SN6_搬入(ST04上)" )
   END_RUNG
   RUNG wire#w5
      Contact( "Auto" )
      Contact( "Com_DB".K03.ST04上托盘在席 )
      Contact( "ST04上阻挡下到位" )
      Contact( "Com_DB".K03.ST05上托盘离席 )
      Contact( "ST05上阻挡上到位" )
      I_Contact( "SN7_搬出(ST05上)" )
      S_Coil( "SN6_搬出(ST04上)" )
   END_RUNG
   RUNG wire#w5
      Contact( "Com_DB".K03.ST04上托盘离席 )
      Contact( "Com_DB".K03.ST05上托盘在席 )
      R_Coil( "SN6_搬出(ST04上)" )
   END_RUNG
   RUNG wire#powerrail
      Contact( "常ON" )
      wire#w6
      P_Contact(operand := "SN6_搬出(ST04上)", bit := #M_Pluse[5])
      S_Coil( "SN7_搬入(ST05上)" )
   END_RUNG
   RUNG wire#w6
      Contact( "Com_DB".K03.ST05上托盘在席 )
      Contact( "ST05上阻挡上到位" )
      R_Coil( "SN7_搬入(ST05上)" )
   END_RUNG
   RUNG wire#w6
      Contact( "Auto" )
      Contact( "Com_DB".K03.ST05上托盘在席 )
      Contact( "ST05上阻挡下到位" )
      Contact( "Com_DB".K03.ST06上托盘离席 )
      Contact( "ST06上阻挡上到位" )
      I_Contact( "SN8_搬出(ST06上)" )
      S_Coil( "SN7_搬出(ST05上)" )
   END_RUNG
   RUNG wire#w6
      Contact( "Com_DB".K03.ST05上托盘离席 )
      Contact( "Com_DB".K03.ST06上托盘在席 )
      R_Coil( "SN7_搬出(ST05上)" )
   END_RUNG
   RUNG wire#powerrail
      Contact( "常ON" )
      wire#w7
      P_Contact(operand := "SN7_搬出(ST05上)", bit := #M_Pluse[6])
      S_Coil( "SN8_搬入(ST06上)" )
   END_RUNG
   RUNG wire#w7
      Contact( "Com_DB".K03.ST06上托盘在席 )
      Contact( "ST06上阻挡上到位" )
      R_Coil( "SN8_搬入(ST06上)" )
   END_RUNG
   RUNG wire#w7
      Contact( "Auto" )
      Contact( "Com_DB".K03.ST06上托盘在席 )
      Contact( "ST06上阻挡下到位" )
      Contact( "Com_DB".K03.ST07上托盘离席 )
      Contact( "ST07上阻挡上到位" )
      I_Contact( "SN9_搬出(ST07上)" )
      S_Coil( "SN8_搬出(ST06上)" )
   END_RUNG
   RUNG wire#w7
      Contact( "Com_DB".K03.ST06上托盘离席 )
      Contact( "Com_DB".K03.ST07上托盘在席 )
      R_Coil( "SN8_搬出(ST06上)" )
   END_RUNG
   RUNG wire#powerrail
      Contact( "常ON" )
      wire#w8
      P_Contact(operand := "SN8_搬出(ST06上)", bit := #M_Pluse[7])
      S_Coil( "SN9_搬入(ST07上)" )
   END_RUNG
   RUNG wire#w8
      Contact( "Com_DB".K03.ST07上托盘在席 )
      Contact( "ST07上阻挡上到位" )
      R_Coil( "SN9_搬入(ST07上)" )
   END_RUNG
   RUNG wire#w8
      Contact( "Auto" )
      Contact( "Com_DB".K03.ST07上托盘在席 )
      Contact( "ST07上阻挡下到位" )
      Contact( "Com_DB".K03.ST08上托盘离席 )
      Contact( "ST08上阻挡上到位" )
      I_Contact( "SN10_搬出(ST08上)" )
      S_Coil( "SN9_搬出(ST07上)" )
   END_RUNG
   RUNG wire#w8
      Contact( "Com_DB".K03.ST07上托盘离席 )
      Contact( "Com_DB".K03.ST08上托盘在席 )
      R_Coil( "SN9_搬出(ST07上)" )
   END_RUNG
   RUNG wire#powerrail
      Contact( "常ON" )
      wire#w9
      P_Contact(operand := "SN9_搬出(ST07上)", bit := #M_Pluse[8])
      S_Coil( "SN10_搬入(ST08上)" )
   END_RUNG
   RUNG wire#w9
      Contact( "Com_DB".K03.ST08上托盘在席 )
      Contact( "ST08上阻挡上到位" )
      R_Coil( "SN10_搬入(ST08上)" )
   END_RUNG
   RUNG wire#w9
      Contact( "Auto" )
      Contact( "Com_DB".K03.ST08上托盘在席 )
      Contact( "ST08上阻挡下到位" )
      Contact( "Com_DB".K03.ST09上托盘离席 )
      Contact( "ST09上阻挡上到位" )
      I_Contact( "SN11_搬出(ST09上)" )
      S_Coil( "SN10_搬出(ST08上)" )
   END_RUNG
   RUNG wire#w9
      Contact( "Com_DB".K03.ST08上托盘离席 )
      Contact( "Com_DB".K03.ST09上托盘在席 )
      R_Coil( "SN10_搬出(ST08上)" )
   END_RUNG
   RUNG wire#powerrail
      Contact( "常ON" )
      wire#w10
      P_Contact(operand := "SN10_搬出(ST08上)", bit := #M_Pluse[9])
      S_Coil( "SN11_搬入(ST09上)" )
   END_RUNG
   RUNG wire#w10
      Contact( "Com_DB".K03.ST09上托盘在席 )
      Contact( "ST09上阻挡上到位" )
      R_Coil( "SN11_搬入(ST09上)" )
   END_RUNG
   RUNG wire#w10
      Contact( "Auto" )
      Contact( "Com_DB".K03.ST09上托盘在席 )
      Contact( "ST09上阻挡下到位" )
      Contact( "Com_DB".K03.EX_托盘离席 )
      Contact( "EX_阻挡上到位" )
      I_Contact( "SN2_搬出(出口)" )
      S_Coil( "SN11_搬出(ST09上)" )
   END_RUNG
   RUNG wire#w10
      Contact( "Com_DB".K03.ST09上托盘离席 )
      Contact( "Com_DB".K03.EX_托盘在席 )
      R_Coil( "SN11_搬出(ST09上)" )
   END_RUNG
   RUNG wire#powerrail
      I_Contact( "常ON" )
      wire#w11
      P_Contact(operand := "SN11_搬出(ST09上)", bit := #M_Pluse[10])
      S_Coil( "SN2_搬入(出口)" )
   END_RUNG
   RUNG wire#w11
      Contact( "Com_DB".K03.EX_托盘在席 )
      Contact( "ST10上阻挡上到位" )
      R_Coil( "SN2_搬入(出口)" )
   END_RUNG
   RUNG wire#w11
      Contact( "Auto" )
      Contact( "Com_DB".K03.ST10上托盘在席 )
      Contact( "ST10上阻挡下到位" )
      Contact( "Com_DB".K03.ST11上托盘离席 )
      Contact( "ST11上阻挡上到位" )
      I_Contact( "SN13_搬出(ST11上)" )
      S_Coil( "SN12_搬出(ST10上)" )
   END_RUNG
   RUNG wire#w11
      Contact( "Com_DB".K03.ST10上托盘离席 )
      Contact( "Com_DB".K03.ST11上托盘在席 )
      R_Coil( "SN12_搬出(ST10上)" )
   END_RUNG
   RUNG wire#powerrail
      I_Contact( "常ON" )
      wire#w12
      P_Contact(operand := "SN12_搬出(ST10上)", bit := #M_Pluse[11])
      S_Coil( "SN13_搬入(ST11上)" )
   END_RUNG
   RUNG wire#w12
      Contact( "Com_DB".K03.ST11上托盘在席 )
      Contact( "ST11上阻挡上到位" )
      R_Coil( "SN13_搬入(ST11上)" )
   END_RUNG
   RUNG wire#w12
      Contact( "Auto" )
      Contact( "Com_DB".K03.ST11上托盘在席 )
      Contact( "ST11上阻挡下到位" )
      Contact( "Com_DB".K03.ST12上托盘离席 )
      Contact( "ST12上阻挡上到位" )
      I_Contact( "SN14_搬出(ST12上)" )
      S_Coil( "SN13_搬出(ST11上)" )
   END_RUNG
   RUNG wire#w12
      Contact( "Com_DB".K03.ST11上托盘离席 )
      Contact( "Com_DB".K03.ST12上托盘在席 )
      R_Coil( "SN13_搬出(ST11上)" )
   END_RUNG
   RUNG wire#powerrail
      I_Contact( "常ON" )
      wire#w13
      P_Contact(operand := "SN13_搬出(ST11上)", bit := #M_Pluse[12])
      S_Coil( "SN14_搬入(ST12上)" )
   END_RUNG
   RUNG wire#w13
      Contact( "Com_DB".K03.ST12上托盘在席 )
      Contact( "ST12上阻挡上到位" )
      R_Coil( "SN14_搬入(ST12上)" )
   END_RUNG
   RUNG wire#w13
      Contact( "Auto" )
      Contact( "Com_DB".K03.ST12上托盘在席 )
      Contact( "ST12上阻挡下到位" )
      Contact( "Com_DB".K03.ST12上托盘离席 )
      Contact( "Com_DB".K03.EX_托盘在席 )
      Contact( "EX_阻挡上到位" )
      I_Contact( "SN2_搬出(出口)" )
      S_Coil( "SN14_搬出(ST12上)" )
   END_RUNG
   RUNG wire#w13
      Contact( "Com_DB".K03.ST12上托盘离席 )
      Contact( "Com_DB".K03.EX_托盘在席 )
      R_Coil( "SN14_搬出(ST12上)" )
   END_RUNG
   RUNG wire#powerrail
      Contact( "常ON" )
      wire#w14
      Contact( "Auto" )
      Contact( "Com_DB".K03.EX_托盘离席 )
      Contact( "EX_提升机上到位" )
      Contact( "EN_阻挡下到位" )
      Contact( "EX_INV2反转" )
      Contact( "Com_DB".K03.ST09上托盘在席 )
      Contact( "ST09上阻挡上到位" )
      I_Contact( "SN11_搬入(ST09上)" )
      S_Coil( "SN2_搬入(出口)" )
   END_RUNG
   RUNG wire#w14
      Contact( "Com_DB".K03.EX_托盘在席 )
      Contact( "EX_阻挡上到位" )
      Contact( "Com_DB".K03.ST09上托盘离席 )
      Contact( "EX_阻挡上到位" )
      R_Coil( "SN2_搬入(出口)" )
   END_RUNG
   RUNG wire#w14
      Contact( "Auto" )
      Contact( "Com_DB".K03.EX_托盘在席 )
      Contact( "EX_提升机下到位" )
      Contact( "EX_阻挡下到位" )
      Contact( "EX_INV2正转" )
      Contact( "Com_DB".K03.ST03下托盘离席 )
      Contact( "ST03下阻挡上到位" )
      I_Contact( "SN15_搬出" )
      S_Coil( "SN2_搬出(出口)" )
   END_RUNG
   RUNG wire#w14
      Contact( "Com_DB".K03.EX_托盘离席 )
      Contact( "EX_阻挡上到位" )
      R_Coil( "SN2_搬出(出口)" )
   END_RUNG
   RUNG wire#powerrail
      Contact( "常ON" )
      wire#w15
      P_Contact(operand := "SN2_搬出(出口)", bit := #M_Pluse[13])
      S_Coil( "SN15_搬入" )
   END_RUNG
   RUNG wire#w15
      Contact( "Com_DB".K03.ST03下托盘在席 )
      Contact( "ST03下阻挡上到位" )
      R_Coil( "SN15_搬入" )
   END_RUNG
   RUNG wire#w15
      Contact( "Auto" )
      Contact( "Com_DB".K03.ST03下托盘在席 )
      Contact( "ST03下阻挡下到位" )
      Contact( "Com_DB".K03.ST02下托盘离席 )
      Contact( "ST02下阻挡上到位" )
      I_Contact( "SN16_搬出" )
      S_Coil( "SN15_搬出" )
   END_RUNG
   RUNG wire#w15
      Contact( "Com_DB".K03.ST03下托盘离席 )
      Contact( "Com_DB".K03.ST02下托盘在席 )
      R_Coil( "SN15_搬出" )
   END_RUNG
   RUNG wire#powerrail
      Contact( "常ON" )
      wire#w16
      P_Contact(operand := "SN15_搬出", bit := #M_Pluse[14])
      S_Coil( "SN16_搬入" )
   END_RUNG
   RUNG wire#w16
      Contact( "Com_DB".K03.ST02下托盘在席 )
      Contact( "ST02下阻挡上到位" )
      R_Coil( "SN16_搬入" )
   END_RUNG
   RUNG wire#w16
      Contact( "Auto" )
      Contact( "Com_DB".K03.ST02下托盘在席 )
      Contact( "ST02下阻挡下到位" )
      Contact( "Com_DB".K03.ST01下托盘离席 )
      Contact( "ST01下阻挡上到位" )
      I_Contact( "SN17_搬出" )
      S_Coil( "SN16_搬出" )
   END_RUNG
   RUNG wire#w16
      Contact( "Com_DB".K03.ST02下托盘离席 )
      Contact( "Com_DB".K03.ST01下托盘在席 )
      R_Coil( "SN16_搬出" )
   END_RUNG
   RUNG wire#powerrail
      Contact( "常ON" )
      wire#w17
      P_Contact(operand := "SN16_搬出", bit := #M_Pluse[15])
      S_Coil( "SN17_搬入" )
   END_RUNG
   RUNG wire#w17
      Contact( "Com_DB".K03.ST01下托盘在席 )
      Contact( "ST01下阻挡上到位" )
      R_Coil( "SN17_搬入" )
   END_RUNG
   RUNG wire#w17
      Contact( "Auto" )
      Contact( "Com_DB".K03.ST01下托盘在席 )
      Contact( "ST01下阻挡下到位" )
      Contact( "Com_DB".K03.EN_托盘离席 )
      Contact( "EN_提升机下到位" )
      Contact( "EN_阻挡下到位" )
      I_Contact( "SN1_搬出(入口)" )
      S_Coil( "SN17_搬出" )
   END_RUNG
   RUNG wire#w17
      Contact( "Com_DB".K03.ST02下托盘离席 )
      Contact( "Com_DB".K03.EN_托盘在席 )
      R_Coil( "SN17_搬出" )
   END_RUNG
   // the same network as SCL:
   IF "常ON" AND "Auto" AND "Com_DB".K03.EN_托盘离席 AND "EN_提升机下到位" AND "EN_阻挡下到位" AND "EN_INV1反转" AND "Com_DB".K03.ST01下托盘在席 AND "ST01下阻挡上到位" AND NOT "SN17_搬入" THEN
       "SN1_搬入(入口)" := TRUE;
   END_IF;
   IF "常ON" AND "Com_DB".K03.EN_托盘在席 AND "EN_阻挡上到位" THEN "SN1_搬入(入口)" := FALSE; END_IF;
   IF "常ON" AND "Auto" AND "Com_DB".K03.EN_托盘在席 AND "EN_提升机上到位" AND "EN_阻挡下到位" AND "EN_INV1正转" AND "Com_DB".K03.ST01上托盘离席 AND "ST01上阻挡上到位" AND NOT "SN3_搬出(ST01上)" THEN
       "SN1_搬出(入口)" := TRUE;
   END_IF;
   IF "常ON" AND "Com_DB".K03.EN_托盘离席 AND "Com_DB".K03.ST01上托盘在席 THEN "SN1_搬出(入口)" := FALSE; END_IF;
   #_w1 := "常ON" AND "SN1_搬出(入口)" AND NOT #M_Pluse[1];   // rising edge of "SN1_搬出(入口)"
   #M_Pluse[1] := "SN1_搬出(入口)";
   IF #_w1 THEN "SN3_搬入(ST01上)" := TRUE; END_IF;
   IF "常ON" AND "Com_DB".K03.ST01上托盘在席 AND "ST01上阻挡上到位" THEN "SN3_搬入(ST01上)" := FALSE; END_IF;
   IF "常ON" AND "Auto" AND "Com_DB".K03.ST01上托盘在席 AND "ST01上阻挡下到位" AND "Com_DB".K03.ST02上托盘离席 AND "ST02上阻挡上到位" AND NOT "SN4_搬出(ST02上)" THEN
       "SN3_搬出(ST01上)" := TRUE;
   END_IF;
   IF "常ON" AND "Com_DB".K03.ST01上托盘离席 AND "Com_DB".K03.ST02上托盘在席 THEN "SN3_搬出(ST01上)" := FALSE; END_IF;
   #_w2 := "常ON" AND "SN3_搬出(ST01上)" AND NOT #M_Pluse[2];   // rising edge of "SN3_搬出(ST01上)"
   #M_Pluse[2] := "SN3_搬出(ST01上)";
   IF #_w2 THEN "SN4_搬入(ST02上)" := TRUE; END_IF;
   IF "常ON" AND "Com_DB".K03.ST02上托盘在席 AND "ST02上阻挡上到位" THEN "SN4_搬入(ST02上)" := FALSE; END_IF;
   IF "常ON" AND "Auto" AND "Com_DB".K03.ST02上托盘在席 AND "ST02上阻挡下到位" AND "Com_DB".K03.ST03上托盘离席 AND "ST03上阻挡上到位" AND NOT "SN5_搬出(ST03上)" THEN
       "SN4_搬出(ST02上)" := TRUE;
   END_IF;
   IF "常ON" AND "Com_DB".K03.ST02上托盘离席 AND "Com_DB".K03.ST03上托盘在席 THEN "SN4_搬出(ST02上)" := FALSE; END_IF;
   #_w3 := "常ON" AND "SN4_搬出(ST02上)" AND NOT #M_Pluse[3];   // rising edge of "SN4_搬出(ST02上)"
   #M_Pluse[3] := "SN4_搬出(ST02上)";
   IF #_w3 THEN "SN5_搬入(ST03上)" := TRUE; END_IF;
   IF "常ON" AND "Com_DB".K03.ST03上托盘在席 AND "ST03上阻挡上到位" THEN "SN5_搬入(ST03上)" := FALSE; END_IF;
   IF "常ON" AND "Auto" AND "Com_DB".K03.ST03上托盘在席 AND "ST03上阻挡下到位" AND "Com_DB".K03.ST04上托盘离席 AND "ST04上阻挡上到位" AND NOT "SN6_搬出(ST04上)" THEN
       "SN5_搬出(ST03上)" := TRUE;
   END_IF;
   IF "常ON" AND "Com_DB".K03.ST03上托盘离席 AND "Com_DB".K03.ST04上托盘在席 THEN "SN5_搬出(ST03上)" := FALSE; END_IF;
   #_w4 := "常ON" AND "SN5_搬出(ST03上)" AND NOT #M_Pluse[4];   // rising edge of "SN5_搬出(ST03上)"
   #M_Pluse[4] := "SN5_搬出(ST03上)";
   IF #_w4 THEN "SN6_搬入(ST04上)" := TRUE; END_IF;
   IF "常ON" AND "Com_DB".K03.ST04上托盘在席 AND "ST04上阻挡上到位" THEN "SN6_搬入(ST04上)" := FALSE; END_IF;
   IF "常ON" AND "Auto" AND "Com_DB".K03.ST04上托盘在席 AND "ST04上阻挡下到位" AND "Com_DB".K03.ST05上托盘离席 AND "ST05上阻挡上到位" AND NOT "SN7_搬出(ST05上)" THEN
       "SN6_搬出(ST04上)" := TRUE;
   END_IF;
   IF "常ON" AND "Com_DB".K03.ST04上托盘离席 AND "Com_DB".K03.ST05上托盘在席 THEN "SN6_搬出(ST04上)" := FALSE; END_IF;
   #_w5 := "常ON" AND "SN6_搬出(ST04上)" AND NOT #M_Pluse[5];   // rising edge of "SN6_搬出(ST04上)"
   #M_Pluse[5] := "SN6_搬出(ST04上)";
   IF #_w5 THEN "SN7_搬入(ST05上)" := TRUE; END_IF;
   IF "常ON" AND "Com_DB".K03.ST05上托盘在席 AND "ST05上阻挡上到位" THEN "SN7_搬入(ST05上)" := FALSE; END_IF;
   IF "常ON" AND "Auto" AND "Com_DB".K03.ST05上托盘在席 AND "ST05上阻挡下到位" AND "Com_DB".K03.ST06上托盘离席 AND "ST06上阻挡上到位" AND NOT "SN8_搬出(ST06上)" THEN
       "SN7_搬出(ST05上)" := TRUE;
   END_IF;
   IF "常ON" AND "Com_DB".K03.ST05上托盘离席 AND "Com_DB".K03.ST06上托盘在席 THEN "SN7_搬出(ST05上)" := FALSE; END_IF;
   #_w6 := "常ON" AND "SN7_搬出(ST05上)" AND NOT #M_Pluse[6];   // rising edge of "SN7_搬出(ST05上)"
   #M_Pluse[6] := "SN7_搬出(ST05上)";
   IF #_w6 THEN "SN8_搬入(ST06上)" := TRUE; END_IF;
   IF "常ON" AND "Com_DB".K03.ST06上托盘在席 AND "ST06上阻挡上到位" THEN "SN8_搬入(ST06上)" := FALSE; END_IF;
   IF "常ON" AND "Auto" AND "Com_DB".K03.ST06上托盘在席 AND "ST06上阻挡下到位" AND "Com_DB".K03.ST07上托盘离席 AND "ST07上阻挡上到位" AND NOT "SN9_搬出(ST07上)" THEN
       "SN8_搬出(ST06上)" := TRUE;
   END_IF;
   IF "常ON" AND "Com_DB".K03.ST06上托盘离席 AND "Com_DB".K03.ST07上托盘在席 THEN "SN8_搬出(ST06上)" := FALSE; END_IF;
   #_w7 := "常ON" AND "SN8_搬出(ST06上)" AND NOT #M_Pluse[7];   // rising edge of "SN8_搬出(ST06上)"
   #M_Pluse[7] := "SN8_搬出(ST06上)";
   IF #_w7 THEN "SN9_搬入(ST07上)" := TRUE; END_IF;
   IF "常ON" AND "Com_DB".K03.ST07上托盘在席 AND "ST07上阻挡上到位" THEN "SN9_搬入(ST07上)" := FALSE; END_IF;
   IF "常ON" AND "Auto" AND "Com_DB".K03.ST07上托盘在席 AND "ST07上阻挡下到位" AND "Com_DB".K03.ST08上托盘离席 AND "ST08上阻挡上到位" AND NOT "SN10_搬出(ST08上)" THEN
       "SN9_搬出(ST07上)" := TRUE;
   END_IF;
   IF "常ON" AND "Com_DB".K03.ST07上托盘离席 AND "Com_DB".K03.ST08上托盘在席 THEN "SN9_搬出(ST07上)" := FALSE; END_IF;
   #_w8 := "常ON" AND "SN9_搬出(ST07上)" AND NOT #M_Pluse[8];   // rising edge of "SN9_搬出(ST07上)"
   #M_Pluse[8] := "SN9_搬出(ST07上)";
   IF #_w8 THEN "SN10_搬入(ST08上)" := TRUE; END_IF;
   IF "常ON" AND "Com_DB".K03.ST08上托盘在席 AND "ST08上阻挡上到位" THEN "SN10_搬入(ST08上)" := FALSE; END_IF;
   IF "常ON" AND "Auto" AND "Com_DB".K03.ST08上托盘在席 AND "ST08上阻挡下到位" AND "Com_DB".K03.ST09上托盘离席 AND "ST09上阻挡上到位" AND NOT "SN11_搬出(ST09上)" THEN
       "SN10_搬出(ST08上)" := TRUE;
   END_IF;
   IF "常ON" AND "Com_DB".K03.ST08上托盘离席 AND "Com_DB".K03.ST09上托盘在席 THEN "SN10_搬出(ST08上)" := FALSE; END_IF;
   #_w9 := "常ON" AND "SN10_搬出(ST08上)" AND NOT #M_Pluse[9];   // rising edge of "SN10_搬出(ST08上)"
   #M_Pluse[9] := "SN10_搬出(ST08上)";
   IF #_w9 THEN "SN11_搬入(ST09上)" := TRUE; END_IF;
   IF "常ON" AND "Com_DB".K03.ST09上托盘在席 AND "ST09上阻挡上到位" THEN "SN11_搬入(ST09上)" := FALSE; END_IF;
   IF "常ON" AND "Auto" AND "Com_DB".K03.ST09上托盘在席 AND "ST09上阻挡下到位" AND "Com_DB".K03.EX_托盘离席 AND "EX_阻挡上到位" AND NOT "SN2_搬出(出口)" THEN
       "SN11_搬出(ST09上)" := TRUE;
   END_IF;
   IF "常ON" AND "Com_DB".K03.ST09上托盘离席 AND "Com_DB".K03.EX_托盘在席 THEN "SN11_搬出(ST09上)" := FALSE; END_IF;
   #_w10 := NOT "常ON" AND "SN11_搬出(ST09上)" AND NOT #M_Pluse[10];   // rising edge of "SN11_搬出(ST09上)"
   #M_Pluse[10] := "SN11_搬出(ST09上)";
   IF #_w10 THEN "SN2_搬入(出口)" := TRUE; END_IF;
   IF NOT "常ON" AND "Com_DB".K03.EX_托盘在席 AND "ST10上阻挡上到位" THEN "SN2_搬入(出口)" := FALSE; END_IF;
   IF NOT "常ON" AND "Auto" AND "Com_DB".K03.ST10上托盘在席 AND "ST10上阻挡下到位" AND "Com_DB".K03.ST11上托盘离席 AND "ST11上阻挡上到位" AND NOT "SN13_搬出(ST11上)" THEN
       "SN12_搬出(ST10上)" := TRUE;
   END_IF;
   IF NOT "常ON" AND "Com_DB".K03.ST10上托盘离席 AND "Com_DB".K03.ST11上托盘在席 THEN "SN12_搬出(ST10上)" := FALSE; END_IF;
   #_w11 := NOT "常ON" AND "SN12_搬出(ST10上)" AND NOT #M_Pluse[11];   // rising edge of "SN12_搬出(ST10上)"
   #M_Pluse[11] := "SN12_搬出(ST10上)";
   IF #_w11 THEN "SN13_搬入(ST11上)" := TRUE; END_IF;
   IF NOT "常ON" AND "Com_DB".K03.ST11上托盘在席 AND "ST11上阻挡上到位" THEN "SN13_搬入(ST11上)" := FALSE; END_IF;
   IF NOT "常ON" AND "Auto" AND "Com_DB".K03.ST11上托盘在席 AND "ST11上阻挡下到位" AND "Com_DB".K03.ST12上托盘离席 AND "ST12上阻挡上到位" AND NOT "SN14_搬出(ST12上)" THEN
       "SN13_搬出(ST11上)" := TRUE;
   END_IF;
   IF NOT "常ON" AND "Com_DB".K03.ST11上托盘离席 AND "Com_DB".K03.ST12上托盘在席 THEN "SN13_搬出(ST11上)" := FALSE; END_IF;
   #_w12 := NOT "常ON" AND "SN13_搬出(ST11上)" AND NOT #M_Pluse[12];   // rising edge of "SN13_搬出(ST11上)"
   #M_Pluse[12] := "SN13_搬出(ST11上)";
   IF #_w12 THEN "SN14_搬入(ST12上)" := TRUE; END_IF;
   IF NOT "常ON" AND "Com_DB".K03.ST12上托盘在席 AND "ST12上阻挡上到位" THEN "SN14_搬入(ST12上)" := FALSE; END_IF;
   IF NOT "常ON" AND "Auto" AND "Com_DB".K03.ST12上托盘在席 AND "ST12上阻挡下到位" AND "Com_DB".K03.ST12上托盘离席 AND "Com_DB".K03.EX_托盘在席 AND "EX_阻挡上到位" AND NOT "SN2_搬出(出口)" THEN
       "SN14_搬出(ST12上)" := TRUE;
   END_IF;
   IF NOT "常ON" AND "Com_DB".K03.ST12上托盘离席 AND "Com_DB".K03.EX_托盘在席 THEN "SN14_搬出(ST12上)" := FALSE; END_IF;
   IF "常ON" AND "Auto" AND "Com_DB".K03.EX_托盘离席 AND "EX_提升机上到位" AND "EN_阻挡下到位" AND "EX_INV2反转" AND "Com_DB".K03.ST09上托盘在席 AND "ST09上阻挡上到位" AND NOT "SN11_搬入(ST09上)" THEN
       "SN2_搬入(出口)" := TRUE;
   END_IF;
   IF "常ON" AND "Com_DB".K03.EX_托盘在席 AND "EX_阻挡上到位" AND "Com_DB".K03.ST09上托盘离席 AND "EX_阻挡上到位" THEN
       "SN2_搬入(出口)" := FALSE;
   END_IF;
   IF "常ON" AND "Auto" AND "Com_DB".K03.EX_托盘在席 AND "EX_提升机下到位" AND "EX_阻挡下到位" AND "EX_INV2正转" AND "Com_DB".K03.ST03下托盘离席 AND "ST03下阻挡上到位" AND NOT "SN15_搬出" THEN
       "SN2_搬出(出口)" := TRUE;
   END_IF;
   IF "常ON" AND "Com_DB".K03.EX_托盘离席 AND "EX_阻挡上到位" THEN "SN2_搬出(出口)" := FALSE; END_IF;
   #_w13 := "常ON" AND "SN2_搬出(出口)" AND NOT #M_Pluse[13];   // rising edge of "SN2_搬出(出口)"
   #M_Pluse[13] := "SN2_搬出(出口)";
   IF #_w13 THEN "SN15_搬入" := TRUE; END_IF;
   IF "常ON" AND "Com_DB".K03.ST03下托盘在席 AND "ST03下阻挡上到位" THEN "SN15_搬入" := FALSE; END_IF;
   IF "常ON" AND "Auto" AND "Com_DB".K03.ST03下托盘在席 AND "ST03下阻挡下到位" AND "Com_DB".K03.ST02下托盘离席 AND "ST02下阻挡上到位" AND NOT "SN16_搬出" THEN
       "SN15_搬出" := TRUE;
   END_IF;
   IF "常ON" AND "Com_DB".K03.ST03下托盘离席 AND "Com_DB".K03.ST02下托盘在席 THEN "SN15_搬出" := FALSE; END_IF;
   #_w14 := "常ON" AND "SN15_搬出" AND NOT #M_Pluse[14];   // rising edge of "SN15_搬出"
   #M_Pluse[14] := "SN15_搬出";
   IF #_w14 THEN "SN16_搬入" := TRUE; END_IF;
   IF "常ON" AND "Com_DB".K03.ST02下托盘在席 AND "ST02下阻挡上到位" THEN "SN16_搬入" := FALSE; END_IF;
   IF "常ON" AND "Auto" AND "Com_DB".K03.ST02下托盘在席 AND "ST02下阻挡下到位" AND "Com_DB".K03.ST01下托盘离席 AND "ST01下阻挡上到位" AND NOT "SN17_搬出" THEN
       "SN16_搬出" := TRUE;
   END_IF;
   IF "常ON" AND "Com_DB".K03.ST02下托盘离席 AND "Com_DB".K03.ST01下托盘在席 THEN "SN16_搬出" := FALSE; END_IF;
   #_w15 := "常ON" AND "SN16_搬出" AND NOT #M_Pluse[15];   // rising edge of "SN16_搬出"
   #M_Pluse[15] := "SN16_搬出";
   IF #_w15 THEN "SN17_搬入" := TRUE; END_IF;
   IF "常ON" AND "Com_DB".K03.ST01下托盘在席 AND "ST01下阻挡上到位" THEN "SN17_搬入" := FALSE; END_IF;
   IF "常ON" AND "Auto" AND "Com_DB".K03.ST01下托盘在席 AND "ST01下阻挡下到位" AND "Com_DB".K03.EN_托盘离席 AND "EN_提升机下到位" AND "EN_阻挡下到位" AND NOT "SN1_搬出(入口)" THEN
       "SN17_搬出" := TRUE;
   END_IF;
   IF "常ON" AND "Com_DB".K03.ST02下托盘离席 AND "Com_DB".K03.EN_托盘在席 THEN "SN17_搬出" := FALSE; END_IF;
END_REGION

REGION Network 26: ST01-ST12放行标志
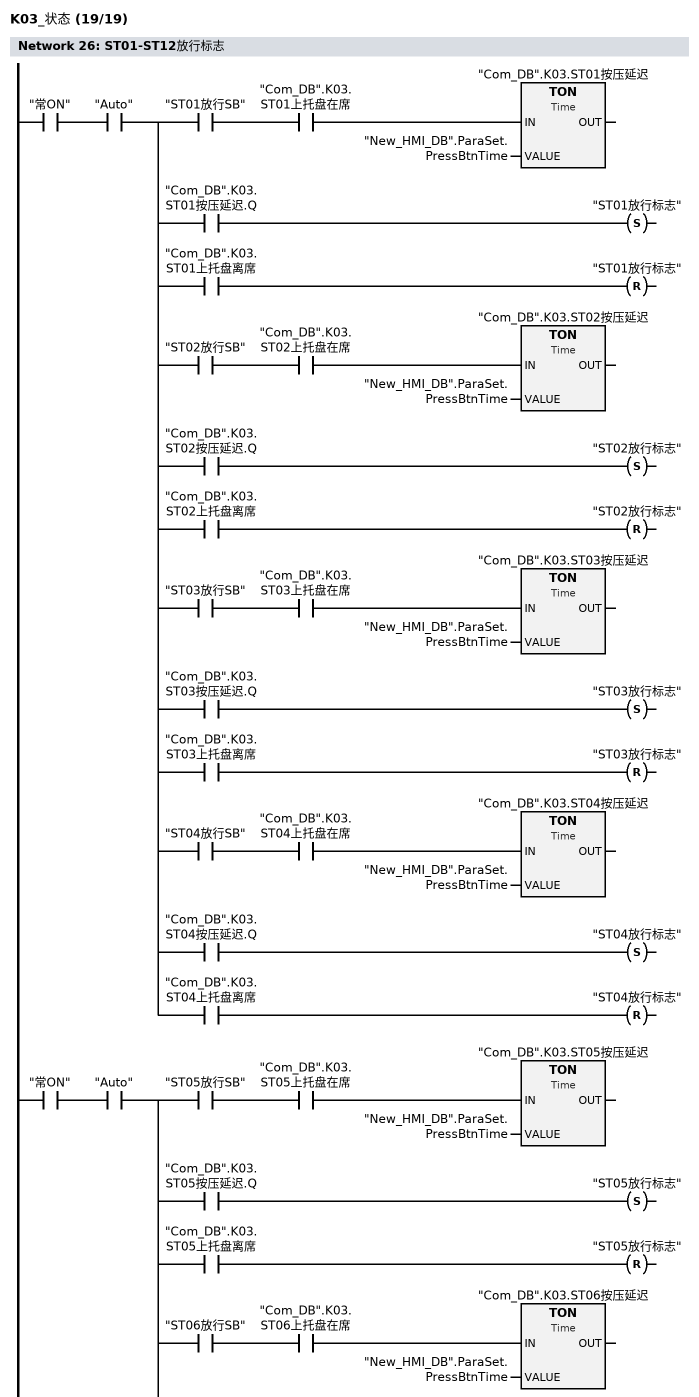
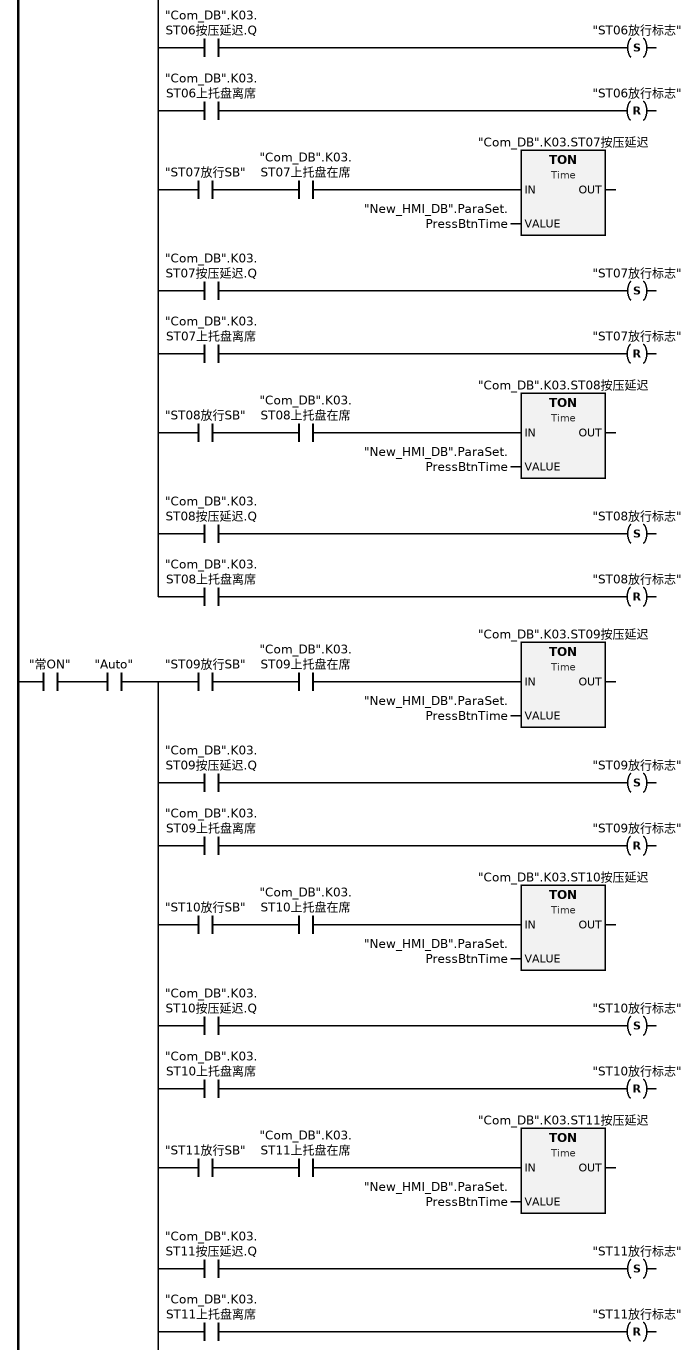
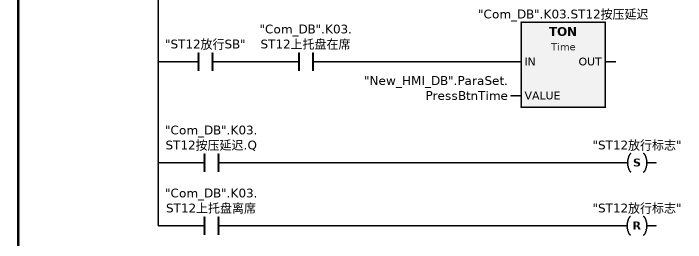
   #_w1 := "常ON" AND "Auto";
   "Com_DB".K03.ST01按压延迟.TON(IN := #_w1 AND "ST01放行SB" AND "Com_DB".K03.ST01上托盘在席, PT := "New_HMI_DB".ParaSet.PressBtnTime);   // TON coil
   IF #_w1 AND "Com_DB".K03.ST01按压延迟.Q THEN "ST01放行标志" := TRUE; END_IF;
   IF #_w1 AND "Com_DB".K03.ST01上托盘离席 THEN "ST01放行标志" := FALSE; END_IF;
   "Com_DB".K03.ST02按压延迟.TON(IN := #_w1 AND "ST02放行SB" AND "Com_DB".K03.ST02上托盘在席, PT := "New_HMI_DB".ParaSet.PressBtnTime);   // TON coil
   IF #_w1 AND "Com_DB".K03.ST02按压延迟.Q THEN "ST02放行标志" := TRUE; END_IF;
   IF #_w1 AND "Com_DB".K03.ST02上托盘离席 THEN "ST02放行标志" := FALSE; END_IF;
   "Com_DB".K03.ST03按压延迟.TON(IN := #_w1 AND "ST03放行SB" AND "Com_DB".K03.ST03上托盘在席, PT := "New_HMI_DB".ParaSet.PressBtnTime);   // TON coil
   IF #_w1 AND "Com_DB".K03.ST03按压延迟.Q THEN "ST03放行标志" := TRUE; END_IF;
   IF #_w1 AND "Com_DB".K03.ST03上托盘离席 THEN "ST03放行标志" := FALSE; END_IF;
   "Com_DB".K03.ST04按压延迟.TON(IN := #_w1 AND "ST04放行SB" AND "Com_DB".K03.ST04上托盘在席, PT := "New_HMI_DB".ParaSet.PressBtnTime);   // TON coil
   IF #_w1 AND "Com_DB".K03.ST04按压延迟.Q THEN "ST04放行标志" := TRUE; END_IF;
   IF #_w1 AND "Com_DB".K03.ST04上托盘离席 THEN "ST04放行标志" := FALSE; END_IF;
   #_w2 := "常ON" AND "Auto";
   "Com_DB".K03.ST05按压延迟.TON(IN := #_w2 AND "ST05放行SB" AND "Com_DB".K03.ST05上托盘在席, PT := "New_HMI_DB".ParaSet.PressBtnTime);   // TON coil
   IF #_w2 AND "Com_DB".K03.ST05按压延迟.Q THEN "ST05放行标志" := TRUE; END_IF;
   IF #_w2 AND "Com_DB".K03.ST05上托盘离席 THEN "ST05放行标志" := FALSE; END_IF;
   "Com_DB".K03.ST06按压延迟.TON(IN := #_w2 AND "ST06放行SB" AND "Com_DB".K03.ST06上托盘在席, PT := "New_HMI_DB".ParaSet.PressBtnTime);   // TON coil
   IF #_w2 AND "Com_DB".K03.ST06按压延迟.Q THEN "ST06放行标志" := TRUE; END_IF;
   IF #_w2 AND "Com_DB".K03.ST06上托盘离席 THEN "ST06放行标志" := FALSE; END_IF;
   "Com_DB".K03.ST07按压延迟.TON(IN := #_w2 AND "ST07放行SB" AND "Com_DB".K03.ST07上托盘在席, PT := "New_HMI_DB".ParaSet.PressBtnTime);   // TON coil
   IF #_w2 AND "Com_DB".K03.ST07按压延迟.Q THEN "ST07放行标志" := TRUE; END_IF;
   IF #_w2 AND "Com_DB".K03.ST07上托盘离席 THEN "ST07放行标志" := FALSE; END_IF;
   "Com_DB".K03.ST08按压延迟.TON(IN := #_w2 AND "ST08放行SB" AND "Com_DB".K03.ST08上托盘在席, PT := "New_HMI_DB".ParaSet.PressBtnTime);   // TON coil
   IF #_w2 AND "Com_DB".K03.ST08按压延迟.Q THEN "ST08放行标志" := TRUE; END_IF;
   IF #_w2 AND "Com_DB".K03.ST08上托盘离席 THEN "ST08放行标志" := FALSE; END_IF;
   #_w3 := "常ON" AND "Auto";
   "Com_DB".K03.ST09按压延迟.TON(IN := #_w3 AND "ST09放行SB" AND "Com_DB".K03.ST09上托盘在席, PT := "New_HMI_DB".ParaSet.PressBtnTime);   // TON coil
   IF #_w3 AND "Com_DB".K03.ST09按压延迟.Q THEN "ST09放行标志" := TRUE; END_IF;
   IF #_w3 AND "Com_DB".K03.ST09上托盘离席 THEN "ST09放行标志" := FALSE; END_IF;
   "Com_DB".K03.ST10按压延迟.TON(IN := #_w3 AND "ST10放行SB" AND "Com_DB".K03.ST10上托盘在席, PT := "New_HMI_DB".ParaSet.PressBtnTime);   // TON coil
   IF #_w3 AND "Com_DB".K03.ST10按压延迟.Q THEN "ST10放行标志" := TRUE; END_IF;
   IF #_w3 AND "Com_DB".K03.ST10上托盘离席 THEN "ST10放行标志" := FALSE; END_IF;
   "Com_DB".K03.ST11按压延迟.TON(IN := #_w3 AND "ST11放行SB" AND "Com_DB".K03.ST11上托盘在席, PT := "New_HMI_DB".ParaSet.PressBtnTime);   // TON coil
   IF #_w3 AND "Com_DB".K03.ST11按压延迟.Q THEN "ST11放行标志" := TRUE; END_IF;
   IF #_w3 AND "Com_DB".K03.ST11上托盘离席 THEN "ST11放行标志" := FALSE; END_IF;
   "Com_DB".K03.ST12按压延迟.TON(IN := #_w3 AND "ST12放行SB" AND "Com_DB".K03.ST12上托盘在席, PT := "New_HMI_DB".ParaSet.PressBtnTime);   // TON coil
   IF #_w3 AND "Com_DB".K03.ST12按压延迟.Q THEN "ST12放行标志" := TRUE; END_IF;
   IF #_w3 AND "Com_DB".K03.ST12上托盘离席 THEN "ST12放行标志" := FALSE; END_IF;
END_REGION
END_FUNCTION_BLOCK
